(* IEC 61131-3 sources: scada_scout/plc_programs (part 2) *)

(* ---- PRG_GPS01GPC02UPM01FCB02.st ---- *)
(* ========================================================================
   PLC PROGRAM: PRG_GPS01GPC02UPM01FCB02
   IED: GPS01GPC02UPM01FCB02
   Device: GPS01GPC02UPM01FCB02
   Generated: 2026-02-05 10:47:33

   This program runs cyclically (default 100ms) and has access to all
   data points of the associated IEC 61850 device. Users can add custom
   logic in the designated sections below.
   ======================================================================== *)

PROGRAM PRG_GPS01GPC02UPM01FCB02
VAR
    (* ====== System Variables ====== *)
    cycle_count: UDINT := 0;           (* Increments each scan cycle *)
    first_scan: BOOL := TRUE;          (* TRUE only on first execution *)
    scan_time_ms: REAL := 0.0;         (* Last scan time in milliseconds *)

    (* ====== IED Connection Status ====== *)
    ied_connected: BOOL := FALSE;      (* TRUE when IED server is running *)
    ied_name: STRING := 'GPS01GPC02UPM01FCB02';
    device_name: STRING := 'GPS01GPC02UPM01FCB02';

    (* ====== Logical Devices ====== *)
    (* Available LDs: AnUn_ArcProtInput1, Application, BinIO, BinIO_BinaryInputs, BinIO_BinaryOutputs, CB1, CB1_Fundamental, Ds1, Ds2, Mod1, Mod1_Channel1, Mod2, Mod2_Channel1, Mod3, Mod3_Channel1, PowS, PowS_MeasPointI3ph1, PowS_MeasPointV3ph1, Rec, Rec_FaultRecorder, VI3p1, VI3p1_5051NOCgndB1, VI3p1_5051OC3phase1, VI3p1_ArcProtection1, VI3p1_Energy, VI3p1_FundSymComp, VI3p1_OperationalValues, VI3p1_ProcessMonitor, VI3p1_ExternalTrip1, VI3p1_67DirOC3phB1, VI3p1_67NDirOCgndB1, ComSupervision, ComSupervision_GOOSE *)

    (* ====== User Variables ====== *)
    (* Add your custom variables here *)
    (* Example:
    timer1: TON;
    counter: INT := 0;
    status_word: WORD;
    *)

END_VAR

(* ======================================================================
   INITIALIZATION SECTION
   Runs once on first scan. Use for setup and initialization.
   ====================================================================== *)
IF first_scan THEN
    (* Initialize user variables here *)
    cycle_count := 0;

    (* Log program start *)
    (* SCADA_LOG('INFO', CONCAT('PLC Program started: ', device_name)); *)

    first_scan := FALSE;
END_IF;

(* ======================================================================
   MAIN CYCLIC EXECUTION
   This section runs continuously every scan cycle (default 100ms).
   ====================================================================== *)

(* Increment cycle counter *)
cycle_count := cycle_count + 1;

(* ====== USER LOGIC SECTION 1: Pre-Processing ====== *)
(* Add logic that should run before main processing *)
(* Example:
IF ied_connected THEN
    (* Read IED data points *)
    (* status_word := READ_IED_DATA(device_name, 'LD0/MMXU1$MX$TotW$mag'); *)
END_IF;
*)

(* ====== USER LOGIC SECTION 2: Main Processing ====== *)
(* Add your main control logic here *)
(* Example:
IF counter > 100 THEN
    counter := 0;
    (* Perform periodic action *)
END_IF;
counter := counter + 1;
*)

(* ====== USER LOGIC SECTION 3: Post-Processing ====== *)
(* Add logic for outputs, writes, and cleanup *)
(* Example:
IF ied_connected THEN
    (* Write control commands to IED *)
    (* WRITE_IED_CONTROL(device_name, 'LD0/CSWI1$CO$Pos', TRUE); *)
END_IF;
*)

(* ====== Built-in Functions Available ====== *)
(*
   READ_IED_DATA(device: STRING, ref: STRING): ANY
       - Read data from IED object reference
       - Example: READ_IED_DATA('MyIED', 'LD0/MMXU1$MX$TotW$mag')

   WRITE_IED_DATA(device: STRING, ref: STRING, value: ANY): BOOL
       - Write data to IED object reference
       - Returns TRUE on success

   WRITE_IED_CONTROL(device: STRING, ref: STRING, value: ANY): BOOL
       - Send control command to IED
       - Returns TRUE on success

   SCADA_LOG(level: STRING, message: STRING)
       - Log message to event log
       - Levels: 'INFO', 'WARNING', 'ERROR'

   GET_DEVICE_STATUS(device: STRING): BOOL
       - Check if device is connected
*)

END_PROGRAM

(* ---- PRG_GPS01GPC02UPM01MCB01.st ---- *)
(* ========================================================================
   PLC PROGRAM: PRG_GPS01GPC02UPM01MCB01
   IED: GPS01GPC02UPM01MCB01
   Device: GPS01GPC02UPM01MCB01
   Generated: 2026-02-05 10:47:34

   This program runs cyclically (default 100ms) and has access to all
   data points of the associated IEC 61850 device. Users can add custom
   logic in the designated sections below.
   ======================================================================== *)

PROGRAM PRG_GPS01GPC02UPM01MCB01
VAR
    (* ====== System Variables ====== *)
    cycle_count: UDINT := 0;           (* Increments each scan cycle *)
    first_scan: BOOL := TRUE;          (* TRUE only on first execution *)
    scan_time_ms: REAL := 0.0;         (* Last scan time in milliseconds *)

    (* ====== IED Connection Status ====== *)
    ied_connected: BOOL := FALSE;      (* TRUE when IED server is running *)
    ied_name: STRING := 'GPS01GPC02UPM01MCB01';
    device_name: STRING := 'GPS01GPC02UPM01MCB01';

    (* ====== Logical Devices ====== *)
    (* Available LDs: AnUn_ArcProtInput1, Application, BinIO, BinIO_BinaryInputs, BinIO_BinaryOutputs, CB1, CB1_Fundamental, Ds1, Ds2, Mod1, Mod1_Channel1, Mod2, Mod2_Channel1, Mod3, Mod3_Channel1, PowS, PowS_MeasPointI3ph1, PowS_MeasPointV3ph1, Rec, Rec_FaultRecorder, VI3p1, VI3p1_5051NOCgndB1, VI3p1_5051OC3phase1, VI3p1_ArcProtection1, VI3p1_Energy, VI3p1_FundSymComp, VI3p1_OperationalValues, VI3p1_ProcessMonitor, VI3p1_ExternalTrip1, VI3p1_67DirOC3phB1, VI3p1_67NDirOCgndB1, VI3p1_ExternalTrip2, ComSupervision, ComSupervision_GOOSE *)

    (* ====== User Variables ====== *)
    (* Add your custom variables here *)
    (* Example:
    timer1: TON;
    counter: INT := 0;
    status_word: WORD;
    *)

END_VAR

(* ======================================================================
   INITIALIZATION SECTION
   Runs once on first scan. Use for setup and initialization.
   ====================================================================== *)
IF first_scan THEN
    (* Initialize user variables here *)
    cycle_count := 0;

    (* Log program start *)
    (* SCADA_LOG('INFO', CONCAT('PLC Program started: ', device_name)); *)

    first_scan := FALSE;
END_IF;

(* ======================================================================
   MAIN CYCLIC EXECUTION
   This section runs continuously every scan cycle (default 100ms).
   ====================================================================== *)

(* Increment cycle counter *)
cycle_count := cycle_count + 1;

(* ====== USER LOGIC SECTION 1: Pre-Processing ====== *)
(* Add logic that should run before main processing *)
(* Example:
IF ied_connected THEN
    (* Read IED data points *)
    (* status_word := READ_IED_DATA(device_name, 'LD0/MMXU1$MX$TotW$mag'); *)
END_IF;
*)

(* ====== USER LOGIC SECTION 2: Main Processing ====== *)
(* Add your main control logic here *)
(* Example:
IF counter > 100 THEN
    counter := 0;
    (* Perform periodic action *)
END_IF;
counter := counter + 1;
*)

(* ====== USER LOGIC SECTION 3: Post-Processing ====== *)
(* Add logic for outputs, writes, and cleanup *)
(* Example:
IF ied_connected THEN
    (* Write control commands to IED *)
    (* WRITE_IED_CONTROL(device_name, 'LD0/CSWI1$CO$Pos', TRUE); *)
END_IF;
*)

(* ====== Built-in Functions Available ====== *)
(*
   READ_IED_DATA(device: STRING, ref: STRING): ANY
       - Read data from IED object reference
       - Example: READ_IED_DATA('MyIED', 'LD0/MMXU1$MX$TotW$mag')

   WRITE_IED_DATA(device: STRING, ref: STRING, value: ANY): BOOL
       - Write data to IED object reference
       - Returns TRUE on success

   WRITE_IED_CONTROL(device: STRING, ref: STRING, value: ANY): BOOL
       - Send control command to IED
       - Returns TRUE on success

   SCADA_LOG(level: STRING, message: STRING)
       - Log message to event log
       - Levels: 'INFO', 'WARNING', 'ERROR'

   GET_DEVICE_STATUS(device: STRING): BOOL
       - Check if device is connected
*)

END_PROGRAM

(* ---- PRG_GPS01GPC03UPM01FCB01.st ---- *)
(* ========================================================================
   PLC PROGRAM: PRG_GPS01GPC03UPM01FCB01
   IED: GPS01GPC03UPM01FCB01
   Device: GPS01GPC03UPM01FCB01
   Generated: 2026-02-05 10:47:34

   This program runs cyclically (default 100ms) and has access to all
   data points of the associated IEC 61850 device. Users can add custom
   logic in the designated sections below.
   ======================================================================== *)

PROGRAM PRG_GPS01GPC03UPM01FCB01
VAR
    (* ====== System Variables ====== *)
    cycle_count: UDINT := 0;           (* Increments each scan cycle *)
    first_scan: BOOL := TRUE;          (* TRUE only on first execution *)
    scan_time_ms: REAL := 0.0;         (* Last scan time in milliseconds *)

    (* ====== IED Connection Status ====== *)
    ied_connected: BOOL := FALSE;      (* TRUE when IED server is running *)
    ied_name: STRING := 'GPS01GPC03UPM01FCB01';
    device_name: STRING := 'GPS01GPC03UPM01FCB01';

    (* ====== Logical Devices ====== *)
    (* Available LDs: AnUn_ArcProtInput1, Application, BinIO, BinIO_BinaryInputs, BinIO_BinaryOutputs, CB1, CB1_Fundamental, Ds1, Ds2, Mod1, Mod1_Channel1, Mod2, Mod2_Channel1, Mod3, Mod3_Channel1, PowS, PowS_MeasPointI3ph1, PowS_MeasPointV3ph1, Rec, Rec_FaultRecorder, VI3p1, VI3p1_5051NOCgndB1, VI3p1_5051OC3phase1, VI3p1_ArcProtection1, VI3p1_Energy, VI3p1_FundSymComp, VI3p1_OperationalValues, VI3p1_ProcessMonitor, VI3p1_ExternalTrip1, VI3p1_67DirOC3phB1, VI3p1_67NDirOCgndB1, ComSupervision, ComSupervision_GOOSE *)

    (* ====== User Variables ====== *)
    (* Add your custom variables here *)
    (* Example:
    timer1: TON;
    counter: INT := 0;
    status_word: WORD;
    *)

END_VAR

(* ======================================================================
   INITIALIZATION SECTION
   Runs once on first scan. Use for setup and initialization.
   ====================================================================== *)
IF first_scan THEN
    (* Initialize user variables here *)
    cycle_count := 0;

    (* Log program start *)
    (* SCADA_LOG('INFO', CONCAT('PLC Program started: ', device_name)); *)

    first_scan := FALSE;
END_IF;

(* ======================================================================
   MAIN CYCLIC EXECUTION
   This section runs continuously every scan cycle (default 100ms).
   ====================================================================== *)

(* Increment cycle counter *)
cycle_count := cycle_count + 1;

(* ====== USER LOGIC SECTION 1: Pre-Processing ====== *)
(* Add logic that should run before main processing *)
(* Example:
IF ied_connected THEN
    (* Read IED data points *)
    (* status_word := READ_IED_DATA(device_name, 'LD0/MMXU1$MX$TotW$mag'); *)
END_IF;
*)

(* ====== USER LOGIC SECTION 2: Main Processing ====== *)
(* Add your main control logic here *)
(* Example:
IF counter > 100 THEN
    counter := 0;
    (* Perform periodic action *)
END_IF;
counter := counter + 1;
*)

(* ====== USER LOGIC SECTION 3: Post-Processing ====== *)
(* Add logic for outputs, writes, and cleanup *)
(* Example:
IF ied_connected THEN
    (* Write control commands to IED *)
    (* WRITE_IED_CONTROL(device_name, 'LD0/CSWI1$CO$Pos', TRUE); *)
END_IF;
*)

(* ====== Built-in Functions Available ====== *)
(*
   READ_IED_DATA(device: STRING, ref: STRING): ANY
       - Read data from IED object reference
       - Example: READ_IED_DATA('MyIED', 'LD0/MMXU1$MX$TotW$mag')

   WRITE_IED_DATA(device: STRING, ref: STRING, value: ANY): BOOL
       - Write data to IED object reference
       - Returns TRUE on success

   WRITE_IED_CONTROL(device: STRING, ref: STRING, value: ANY): BOOL
       - Send control command to IED
       - Returns TRUE on success

   SCADA_LOG(level: STRING, message: STRING)
       - Log message to event log
       - Levels: 'INFO', 'WARNING', 'ERROR'

   GET_DEVICE_STATUS(device: STRING): BOOL
       - Check if device is connected
*)

END_PROGRAM

(* ---- PRG_GPS01GPC03UPM01FCB02.st ---- *)
(* ========================================================================
   PLC PROGRAM: PRG_GPS01GPC03UPM01FCB02
   IED: GPS01GPC03UPM01FCB02
   Device: GPS01GPC03UPM01FCB02
   Generated: 2026-02-05 10:47:35

   This program runs cyclically (default 100ms) and has access to all
   data points of the associated IEC 61850 device. Users can add custom
   logic in the designated sections below.
   ======================================================================== *)

PROGRAM PRG_GPS01GPC03UPM01FCB02
VAR
    (* ====== System Variables ====== *)
    cycle_count: UDINT := 0;           (* Increments each scan cycle *)
    first_scan: BOOL := TRUE;          (* TRUE only on first execution *)
    scan_time_ms: REAL := 0.0;         (* Last scan time in milliseconds *)

    (* ====== IED Connection Status ====== *)
    ied_connected: BOOL := FALSE;      (* TRUE when IED server is running *)
    ied_name: STRING := 'GPS01GPC03UPM01FCB02';
    device_name: STRING := 'GPS01GPC03UPM01FCB02';

    (* ====== Logical Devices ====== *)
    (* Available LDs: AnUn_ArcProtInput1, Application, BinIO, BinIO_BinaryInputs, BinIO_BinaryOutputs, CB1, CB1_Fundamental, Ds1, Ds2, Mod1, Mod1_Channel1, Mod2, Mod2_Channel1, Mod3, Mod3_Channel1, PowS, PowS_MeasPointI3ph1, PowS_MeasPointV3ph1, Rec, Rec_FaultRecorder, VI3p1, VI3p1_5051NOCgndB1, VI3p1_5051OC3phase1, VI3p1_ArcProtection1, VI3p1_Energy, VI3p1_FundSymComp, VI3p1_OperationalValues, VI3p1_ProcessMonitor, VI3p1_ExternalTrip1, VI3p1_67DirOC3phB1, VI3p1_67NDirOCgndB1, ComSupervision, ComSupervision_GOOSE *)

    (* ====== User Variables ====== *)
    (* Add your custom variables here *)
    (* Example:
    timer1: TON;
    counter: INT := 0;
    status_word: WORD;
    *)

END_VAR

(* ======================================================================
   INITIALIZATION SECTION
   Runs once on first scan. Use for setup and initialization.
   ====================================================================== *)
IF first_scan THEN
    (* Initialize user variables here *)
    cycle_count := 0;

    (* Log program start *)
    (* SCADA_LOG('INFO', CONCAT('PLC Program started: ', device_name)); *)

    first_scan := FALSE;
END_IF;

(* ======================================================================
   MAIN CYCLIC EXECUTION
   This section runs continuously every scan cycle (default 100ms).
   ====================================================================== *)

(* Increment cycle counter *)
cycle_count := cycle_count + 1;

(* ====== USER LOGIC SECTION 1: Pre-Processing ====== *)
(* Add logic that should run before main processing *)
(* Example:
IF ied_connected THEN
    (* Read IED data points *)
    (* status_word := READ_IED_DATA(device_name, 'LD0/MMXU1$MX$TotW$mag'); *)
END_IF;
*)

(* ====== USER LOGIC SECTION 2: Main Processing ====== *)
(* Add your main control logic here *)
(* Example:
IF counter > 100 THEN
    counter := 0;
    (* Perform periodic action *)
END_IF;
counter := counter + 1;
*)

(* ====== USER LOGIC SECTION 3: Post-Processing ====== *)
(* Add logic for outputs, writes, and cleanup *)
(* Example:
IF ied_connected THEN
    (* Write control commands to IED *)
    (* WRITE_IED_CONTROL(device_name, 'LD0/CSWI1$CO$Pos', TRUE); *)
END_IF;
*)

(* ====== Built-in Functions Available ====== *)
(*
   READ_IED_DATA(device: STRING, ref: STRING): ANY
       - Read data from IED object reference
       - Example: READ_IED_DATA('MyIED', 'LD0/MMXU1$MX$TotW$mag')

   WRITE_IED_DATA(device: STRING, ref: STRING, value: ANY): BOOL
       - Write data to IED object reference
       - Returns TRUE on success

   WRITE_IED_CONTROL(device: STRING, ref: STRING, value: ANY): BOOL
       - Send control command to IED
       - Returns TRUE on success

   SCADA_LOG(level: STRING, message: STRING)
       - Log message to event log
       - Levels: 'INFO', 'WARNING', 'ERROR'

   GET_DEVICE_STATUS(device: STRING): BOOL
       - Check if device is connected
*)

END_PROGRAM

(* ---- PRG_GPS01GPC03UPM01MCB01.st ---- *)
(* ========================================================================
   PLC PROGRAM: PRG_GPS01GPC03UPM01MCB01
   IED: GPS01GPC03UPM01MCB01
   Device: GPS01GPC03UPM01MCB01
   Generated: 2026-02-05 10:47:36

   This program runs cyclically (default 100ms) and has access to all
   data points of the associated IEC 61850 device. Users can add custom
   logic in the designated sections below.
   ======================================================================== *)

PROGRAM PRG_GPS01GPC03UPM01MCB01
VAR
    (* ====== System Variables ====== *)
    cycle_count: UDINT := 0;           (* Increments each scan cycle *)
    first_scan: BOOL := TRUE;          (* TRUE only on first execution *)
    scan_time_ms: REAL := 0.0;         (* Last scan time in milliseconds *)

    (* ====== IED Connection Status ====== *)
    ied_connected: BOOL := FALSE;      (* TRUE when IED server is running *)
    ied_name: STRING := 'GPS01GPC03UPM01MCB01';
    device_name: STRING := 'GPS01GPC03UPM01MCB01';

    (* ====== Logical Devices ====== *)
    (* Available LDs: AnUn_ArcProtInput1, Application, BinIO, BinIO_BinaryInputs, BinIO_BinaryOutputs, CB1, CB1_Fundamental, Ds1, Ds2, Mod1, Mod1_Channel1, Mod2, Mod2_Channel1, Mod3, Mod3_Channel1, PowS, PowS_MeasPointI3ph1, PowS_MeasPointV3ph1, Rec, Rec_FaultRecorder, VI3p1, VI3p1_5051NOCgndB1, VI3p1_5051OC3phase1, VI3p1_ArcProtection1, VI3p1_Energy, VI3p1_FundSymComp, VI3p1_OperationalValues, VI3p1_ProcessMonitor, VI3p1_67DirOC3phB1, VI3p1_ExternalTrip1, VI3p1_67NDirOCgndB1, VI3p1_ExternalTrip2, ComSupervision, ComSupervision_GOOSE *)

    (* ====== User Variables ====== *)
    (* Add your custom variables here *)
    (* Example:
    timer1: TON;
    counter: INT := 0;
    status_word: WORD;
    *)

END_VAR

(* ======================================================================
   INITIALIZATION SECTION
   Runs once on first scan. Use for setup and initialization.
   ====================================================================== *)
IF first_scan THEN
    (* Initialize user variables here *)
    cycle_count := 0;

    (* Log program start *)
    (* SCADA_LOG('INFO', CONCAT('PLC Program started: ', device_name)); *)

    first_scan := FALSE;
END_IF;

(* ======================================================================
   MAIN CYCLIC EXECUTION
   This section runs continuously every scan cycle (default 100ms).
   ====================================================================== *)

(* Increment cycle counter *)
cycle_count := cycle_count + 1;

(* ====== USER LOGIC SECTION 1: Pre-Processing ====== *)
(* Add logic that should run before main processing *)
(* Example:
IF ied_connected THEN
    (* Read IED data points *)
    (* status_word := READ_IED_DATA(device_name, 'LD0/MMXU1$MX$TotW$mag'); *)
END_IF;
*)

(* ====== USER LOGIC SECTION 2: Main Processing ====== *)
(* Add your main control logic here *)
(* Example:
IF counter > 100 THEN
    counter := 0;
    (* Perform periodic action *)
END_IF;
counter := counter + 1;
*)

(* ====== USER LOGIC SECTION 3: Post-Processing ====== *)
(* Add logic for outputs, writes, and cleanup *)
(* Example:
IF ied_connected THEN
    (* Write control commands to IED *)
    (* WRITE_IED_CONTROL(device_name, 'LD0/CSWI1$CO$Pos', TRUE); *)
END_IF;
*)

(* ====== Built-in Functions Available ====== *)
(*
   READ_IED_DATA(device: STRING, ref: STRING): ANY
       - Read data from IED object reference
       - Example: READ_IED_DATA('MyIED', 'LD0/MMXU1$MX$TotW$mag')

   WRITE_IED_DATA(device: STRING, ref: STRING, value: ANY): BOOL
       - Write data to IED object reference
       - Returns TRUE on success

   WRITE_IED_CONTROL(device: STRING, ref: STRING, value: ANY): BOOL
       - Send control command to IED
       - Returns TRUE on success

   SCADA_LOG(level: STRING, message: STRING)
       - Log message to event log
       - Levels: 'INFO', 'WARNING', 'ERROR'

   GET_DEVICE_STATUS(device: STRING): BOOL
       - Check if device is connected
*)

END_PROGRAM

(* ---- PRG_GPS01GPC04UPM01FCB01.st ---- *)
(* ========================================================================
   PLC PROGRAM: PRG_GPS01GPC04UPM01FCB01
   IED: GPS01GPC04UPM01FCB01
   Device: GPS01GPC04UPM01FCB01
   Generated: 2026-02-05 10:47:36

   This program runs cyclically (default 100ms) and has access to all
   data points of the associated IEC 61850 device. Users can add custom
   logic in the designated sections below.
   ======================================================================== *)

PROGRAM PRG_GPS01GPC04UPM01FCB01
VAR
    (* ====== System Variables ====== *)
    cycle_count: UDINT := 0;           (* Increments each scan cycle *)
    first_scan: BOOL := TRUE;          (* TRUE only on first execution *)
    scan_time_ms: REAL := 0.0;         (* Last scan time in milliseconds *)

    (* ====== IED Connection Status ====== *)
    ied_connected: BOOL := FALSE;      (* TRUE when IED server is running *)
    ied_name: STRING := 'GPS01GPC04UPM01FCB01';
    device_name: STRING := 'GPS01GPC04UPM01FCB01';

    (* ====== Logical Devices ====== *)
    (* Available LDs: AnUn_ArcProtInput1, Application, BinIO, BinIO_BinaryInputs, BinIO_BinaryOutputs, CB1, CB1_Fundamental, Ds1, Ds2, Mod1, Mod1_Channel1, Mod2, Mod2_Channel1, Mod3, Mod3_Channel1, PowS, PowS_MeasPointI3ph1, PowS_MeasPointV3ph1, Rec, Rec_FaultRecorder, VI3p1, VI3p1_5051NOCgndB1, VI3p1_5051OC3phase1, VI3p1_ArcProtection1, VI3p1_Energy, VI3p1_FundSymComp, VI3p1_OperationalValues, VI3p1_ProcessMonitor, VI3p1_ExternalTrip1, VI3p1_67DirOC3phB1, VI3p1_67NDirOCgndB1, ComSupervision, ComSupervision_GOOSE *)

    (* ====== User Variables ====== *)
    (* Add your custom variables here *)
    (* Example:
    timer1: TON;
    counter: INT := 0;
    status_word: WORD;
    *)

END_VAR

(* ======================================================================
   INITIALIZATION SECTION
   Runs once on first scan. Use for setup and initialization.
   ====================================================================== *)
IF first_scan THEN
    (* Initialize user variables here *)
    cycle_count := 0;

    (* Log program start *)
    (* SCADA_LOG('INFO', CONCAT('PLC Program started: ', device_name)); *)

    first_scan := FALSE;
END_IF;

(* ======================================================================
   MAIN CYCLIC EXECUTION
   This section runs continuously every scan cycle (default 100ms).
   ====================================================================== *)

(* Increment cycle counter *)
cycle_count := cycle_count + 1;

(* ====== USER LOGIC SECTION 1: Pre-Processing ====== *)
(* Add logic that should run before main processing *)
(* Example:
IF ied_connected THEN
    (* Read IED data points *)
    (* status_word := READ_IED_DATA(device_name, 'LD0/MMXU1$MX$TotW$mag'); *)
END_IF;
*)

(* ====== USER LOGIC SECTION 2: Main Processing ====== *)
(* Add your main control logic here *)
(* Example:
IF counter > 100 THEN
    counter := 0;
    (* Perform periodic action *)
END_IF;
counter := counter + 1;
*)

(* ====== USER LOGIC SECTION 3: Post-Processing ====== *)
(* Add logic for outputs, writes, and cleanup *)
(* Example:
IF ied_connected THEN
    (* Write control commands to IED *)
    (* WRITE_IED_CONTROL(device_name, 'LD0/CSWI1$CO$Pos', TRUE); *)
END_IF;
*)

(* ====== Built-in Functions Available ====== *)
(*
   READ_IED_DATA(device: STRING, ref: STRING): ANY
       - Read data from IED object reference
       - Example: READ_IED_DATA('MyIED', 'LD0/MMXU1$MX$TotW$mag')

   WRITE_IED_DATA(device: STRING, ref: STRING, value: ANY): BOOL
       - Write data to IED object reference
       - Returns TRUE on success

   WRITE_IED_CONTROL(device: STRING, ref: STRING, value: ANY): BOOL
       - Send control command to IED
       - Returns TRUE on success

   SCADA_LOG(level: STRING, message: STRING)
       - Log message to event log
       - Levels: 'INFO', 'WARNING', 'ERROR'

   GET_DEVICE_STATUS(device: STRING): BOOL
       - Check if device is connected
*)

END_PROGRAM

(* ---- PRG_GPS01GPC04UPM01FCB02.st ---- *)
(* ========================================================================
   PLC PROGRAM: PRG_GPS01GPC04UPM01FCB02
   IED: GPS01GPC04UPM01FCB02
   Device: GPS01GPC04UPM01FCB02
   Generated: 2026-02-05 10:47:38

   This program runs cyclically (default 100ms) and has access to all
   data points of the associated IEC 61850 device. Users can add custom
   logic in the designated sections below.
   ======================================================================== *)

PROGRAM PRG_GPS01GPC04UPM01FCB02
VAR
    (* ====== System Variables ====== *)
    cycle_count: UDINT := 0;           (* Increments each scan cycle *)
    first_scan: BOOL := TRUE;          (* TRUE only on first execution *)
    scan_time_ms: REAL := 0.0;         (* Last scan time in milliseconds *)

    (* ====== IED Connection Status ====== *)
    ied_connected: BOOL := FALSE;      (* TRUE when IED server is running *)
    ied_name: STRING := 'GPS01GPC04UPM01FCB02';
    device_name: STRING := 'GPS01GPC04UPM01FCB02';

    (* ====== Logical Devices ====== *)
    (* Available LDs: AnUn_ArcProtInput1, Application, BinIO, BinIO_BinaryInputs, BinIO_BinaryOutputs, CB1, CB1_Fundamental, Ds1, Ds2, Mod1, Mod1_Channel1, Mod2, Mod2_Channel1, Mod3, Mod3_Channel1, PowS, PowS_MeasPointI3ph1, PowS_MeasPointV3ph1, Rec, Rec_FaultRecorder, VI3p1, VI3p1_5051NOCgndB1, VI3p1_5051OC3phase1, VI3p1_ArcProtection1, VI3p1_Energy, VI3p1_FundSymComp, VI3p1_OperationalValues, VI3p1_ProcessMonitor, VI3p1_ExternalTrip1, VI3p1_67DirOC3phB1, VI3p1_67NDirOCgndB1, ComSupervision, ComSupervision_GOOSE *)

    (* ====== User Variables ====== *)
    (* Add your custom variables here *)
    (* Example:
    timer1: TON;
    counter: INT := 0;
    status_word: WORD;
    *)

END_VAR

(* ======================================================================
   INITIALIZATION SECTION
   Runs once on first scan. Use for setup and initialization.
   ====================================================================== *)
IF first_scan THEN
    (* Initialize user variables here *)
    cycle_count := 0;

    (* Log program start *)
    (* SCADA_LOG('INFO', CONCAT('PLC Program started: ', device_name)); *)

    first_scan := FALSE;
END_IF;

(* ======================================================================
   MAIN CYCLIC EXECUTION
   This section runs continuously every scan cycle (default 100ms).
   ====================================================================== *)

(* Increment cycle counter *)
cycle_count := cycle_count + 1;

(* ====== USER LOGIC SECTION 1: Pre-Processing ====== *)
(* Add logic that should run before main processing *)
(* Example:
IF ied_connected THEN
    (* Read IED data points *)
    (* status_word := READ_IED_DATA(device_name, 'LD0/MMXU1$MX$TotW$mag'); *)
END_IF;
*)

(* ====== USER LOGIC SECTION 2: Main Processing ====== *)
(* Add your main control logic here *)
(* Example:
IF counter > 100 THEN
    counter := 0;
    (* Perform periodic action *)
END_IF;
counter := counter + 1;
*)

(* ====== USER LOGIC SECTION 3: Post-Processing ====== *)
(* Add logic for outputs, writes, and cleanup *)
(* Example:
IF ied_connected THEN
    (* Write control commands to IED *)
    (* WRITE_IED_CONTROL(device_name, 'LD0/CSWI1$CO$Pos', TRUE); *)
END_IF;
*)

(* ====== Built-in Functions Available ====== *)
(*
   READ_IED_DATA(device: STRING, ref: STRING): ANY
       - Read data from IED object reference
       - Example: READ_IED_DATA('MyIED', 'LD0/MMXU1$MX$TotW$mag')

   WRITE_IED_DATA(device: STRING, ref: STRING, value: ANY): BOOL
       - Write data to IED object reference
       - Returns TRUE on success

   WRITE_IED_CONTROL(device: STRING, ref: STRING, value: ANY): BOOL
       - Send control command to IED
       - Returns TRUE on success

   SCADA_LOG(level: STRING, message: STRING)
       - Log message to event log
       - Levels: 'INFO', 'WARNING', 'ERROR'

   GET_DEVICE_STATUS(device: STRING): BOOL
       - Check if device is connected
*)

END_PROGRAM

(* ---- PRG_GPS01GPC04UPM01MCB01.st ---- *)
(* ========================================================================
   PLC PROGRAM: PRG_GPS01GPC04UPM01MCB01
   IED: GPS01GPC04UPM01MCB01
   Device: GPS01GPC04UPM01MCB01
   Generated: 2026-02-05 10:47:39

   This program runs cyclically (default 100ms) and has access to all
   data points of the associated IEC 61850 device. Users can add custom
   logic in the designated sections below.
   ======================================================================== *)

PROGRAM PRG_GPS01GPC04UPM01MCB01
VAR
    (* ====== System Variables ====== *)
    cycle_count: UDINT := 0;           (* Increments each scan cycle *)
    first_scan: BOOL := TRUE;          (* TRUE only on first execution *)
    scan_time_ms: REAL := 0.0;         (* Last scan time in milliseconds *)

    (* ====== IED Connection Status ====== *)
    ied_connected: BOOL := FALSE;      (* TRUE when IED server is running *)
    ied_name: STRING := 'GPS01GPC04UPM01MCB01';
    device_name: STRING := 'GPS01GPC04UPM01MCB01';

    (* ====== Logical Devices ====== *)
    (* Available LDs: AnUn_ArcProtInput1, Application, BinIO, BinIO_BinaryInputs, BinIO_BinaryOutputs, CB1, CB1_Fundamental, Ds1, Ds2, Mod1, Mod1_Channel1, Mod2, Mod2_Channel1, Mod3, Mod3_Channel1, PowS, PowS_MeasPointI3ph1, PowS_MeasPointV3ph1, Rec, Rec_FaultRecorder, VI3p1, VI3p1_5051NOCgndB1, VI3p1_5051OC3phase1, VI3p1_ArcProtection1, VI3p1_Energy, VI3p1_FundSymComp, VI3p1_OperationalValues, VI3p1_ProcessMonitor, VI3p1_ExternalTrip1, VI3p1_67DirOC3phB1, VI3p1_67NDirOCgndB1, VI3p1_ExternalTrip2, ComSupervision, ComSupervision_GOOSE *)

    (* ====== User Variables ====== *)
    (* Add your custom variables here *)
    (* Example:
    timer1: TON;
    counter: INT := 0;
    status_word: WORD;
    *)

END_VAR

(* ======================================================================
   INITIALIZATION SECTION
   Runs once on first scan. Use for setup and initialization.
   ====================================================================== *)
IF first_scan THEN
    (* Initialize user variables here *)
    cycle_count := 0;

    (* Log program start *)
    (* SCADA_LOG('INFO', CONCAT('PLC Program started: ', device_name)); *)

    first_scan := FALSE;
END_IF;

(* ======================================================================
   MAIN CYCLIC EXECUTION
   This section runs continuously every scan cycle (default 100ms).
   ====================================================================== *)

(* Increment cycle counter *)
cycle_count := cycle_count + 1;

(* ====== USER LOGIC SECTION 1: Pre-Processing ====== *)
(* Add logic that should run before main processing *)
(* Example:
IF ied_connected THEN
    (* Read IED data points *)
    (* status_word := READ_IED_DATA(device_name, 'LD0/MMXU1$MX$TotW$mag'); *)
END_IF;
*)

(* ====== USER LOGIC SECTION 2: Main Processing ====== *)
(* Add your main control logic here *)
(* Example:
IF counter > 100 THEN
    counter := 0;
    (* Perform periodic action *)
END_IF;
counter := counter + 1;
*)

(* ====== USER LOGIC SECTION 3: Post-Processing ====== *)
(* Add logic for outputs, writes, and cleanup *)
(* Example:
IF ied_connected THEN
    (* Write control commands to IED *)
    (* WRITE_IED_CONTROL(device_name, 'LD0/CSWI1$CO$Pos', TRUE); *)
END_IF;
*)

(* ====== Built-in Functions Available ====== *)
(*
   READ_IED_DATA(device: STRING, ref: STRING): ANY
       - Read data from IED object reference
       - Example: READ_IED_DATA('MyIED', 'LD0/MMXU1$MX$TotW$mag')

   WRITE_IED_DATA(device: STRING, ref: STRING, value: ANY): BOOL
       - Write data to IED object reference
       - Returns TRUE on success

   WRITE_IED_CONTROL(device: STRING, ref: STRING, value: ANY): BOOL
       - Send control command to IED
       - Returns TRUE on success

   SCADA_LOG(level: STRING, message: STRING)
       - Log message to event log
       - Levels: 'INFO', 'WARNING', 'ERROR'

   GET_DEVICE_STATUS(device: STRING): BOOL
       - Check if device is connected
*)

END_PROGRAM

(* ---- PRG_GPS01GPC05UPM01FCB01.st ---- *)
(* ========================================================================
   PLC PROGRAM: PRG_GPS01GPC05UPM01FCB01
   IED: GPS01GPC05UPM01FCB01
   Device: GPS01GPC05UPM01FCB01
   Generated: 2026-02-05 10:47:39

   This program runs cyclically (default 100ms) and has access to all
   data points of the associated IEC 61850 device. Users can add custom
   logic in the designated sections below.
   ======================================================================== *)

PROGRAM PRG_GPS01GPC05UPM01FCB01
VAR
    (* ====== System Variables ====== *)
    cycle_count: UDINT := 0;           (* Increments each scan cycle *)
    first_scan: BOOL := TRUE;          (* TRUE only on first execution *)
    scan_time_ms: REAL := 0.0;         (* Last scan time in milliseconds *)

    (* ====== IED Connection Status ====== *)
    ied_connected: BOOL := FALSE;      (* TRUE when IED server is running *)
    ied_name: STRING := 'GPS01GPC05UPM01FCB01';
    device_name: STRING := 'GPS01GPC05UPM01FCB01';

    (* ====== Logical Devices ====== *)
    (* Available LDs: AnUn_ArcProtInput1, Application, BinIO, BinIO_BinaryInputs, BinIO_BinaryOutputs, CB1, CB1_Fundamental, Ds1, Ds2, Mod1, Mod1_Channel1, Mod2, Mod2_Channel1, Mod3, Mod3_Channel1, PowS, PowS_MeasPointI3ph1, PowS_MeasPointV3ph1, Rec, Rec_FaultRecorder, VI3p1, VI3p1_5051NOCgndB1, VI3p1_5051OC3phase1, VI3p1_ArcProtection1, VI3p1_Energy, VI3p1_FundSymComp, VI3p1_OperationalValues, VI3p1_ProcessMonitor, VI3p1_ExternalTrip1, VI3p1_67DirOC3phB1, VI3p1_67NDirOCgndB1, ComSupervision, ComSupervision_GOOSE *)

    (* ====== User Variables ====== *)
    (* Add your custom variables here *)
    (* Example:
    timer1: TON;
    counter: INT := 0;
    status_word: WORD;
    *)

END_VAR

(* ======================================================================
   INITIALIZATION SECTION
   Runs once on first scan. Use for setup and initialization.
   ====================================================================== *)
IF first_scan THEN
    (* Initialize user variables here *)
    cycle_count := 0;

    (* Log program start *)
    (* SCADA_LOG('INFO', CONCAT('PLC Program started: ', device_name)); *)

    first_scan := FALSE;
END_IF;

(* ======================================================================
   MAIN CYCLIC EXECUTION
   This section runs continuously every scan cycle (default 100ms).
   ====================================================================== *)

(* Increment cycle counter *)
cycle_count := cycle_count + 1;

(* ====== USER LOGIC SECTION 1: Pre-Processing ====== *)
(* Add logic that should run before main processing *)
(* Example:
IF ied_connected THEN
    (* Read IED data points *)
    (* status_word := READ_IED_DATA(device_name, 'LD0/MMXU1$MX$TotW$mag'); *)
END_IF;
*)

(* ====== USER LOGIC SECTION 2: Main Processing ====== *)
(* Add your main control logic here *)
(* Example:
IF counter > 100 THEN
    counter := 0;
    (* Perform periodic action *)
END_IF;
counter := counter + 1;
*)

(* ====== USER LOGIC SECTION 3: Post-Processing ====== *)
(* Add logic for outputs, writes, and cleanup *)
(* Example:
IF ied_connected THEN
    (* Write control commands to IED *)
    (* WRITE_IED_CONTROL(device_name, 'LD0/CSWI1$CO$Pos', TRUE); *)
END_IF;
*)

(* ====== Built-in Functions Available ====== *)
(*
   READ_IED_DATA(device: STRING, ref: STRING): ANY
       - Read data from IED object reference
       - Example: READ_IED_DATA('MyIED', 'LD0/MMXU1$MX$TotW$mag')

   WRITE_IED_DATA(device: STRING, ref: STRING, value: ANY): BOOL
       - Write data to IED object reference
       - Returns TRUE on success

   WRITE_IED_CONTROL(device: STRING, ref: STRING, value: ANY): BOOL
       - Send control command to IED
       - Returns TRUE on success

   SCADA_LOG(level: STRING, message: STRING)
       - Log message to event log
       - Levels: 'INFO', 'WARNING', 'ERROR'

   GET_DEVICE_STATUS(device: STRING): BOOL
       - Check if device is connected
*)

END_PROGRAM

(* ---- PRG_GPS01GPC05UPM01FCB02.st ---- *)
(* ========================================================================
   PLC PROGRAM: PRG_GPS01GPC05UPM01FCB02
   IED: GPS01GPC05UPM01FCB02
   Device: GPS01GPC05UPM01FCB02
   Generated: 2026-02-05 10:47:40

   This program runs cyclically (default 100ms) and has access to all
   data points of the associated IEC 61850 device. Users can add custom
   logic in the designated sections below.
   ======================================================================== *)

PROGRAM PRG_GPS01GPC05UPM01FCB02
VAR
    (* ====== System Variables ====== *)
    cycle_count: UDINT := 0;           (* Increments each scan cycle *)
    first_scan: BOOL := TRUE;          (* TRUE only on first execution *)
    scan_time_ms: REAL := 0.0;         (* Last scan time in milliseconds *)

    (* ====== IED Connection Status ====== *)
    ied_connected: BOOL := FALSE;      (* TRUE when IED server is running *)
    ied_name: STRING := 'GPS01GPC05UPM01FCB02';
    device_name: STRING := 'GPS01GPC05UPM01FCB02';

    (* ====== Logical Devices ====== *)
    (* Available LDs: AnUn_ArcProtInput1, Application, BinIO, BinIO_BinaryInputs, BinIO_BinaryOutputs, CB1, CB1_Fundamental, Ds1, Ds2, Mod1, Mod1_Channel1, Mod2, Mod2_Channel1, Mod3, Mod3_Channel1, PowS, PowS_MeasPointI3ph1, PowS_MeasPointV3ph1, Rec, Rec_FaultRecorder, VI3p1, VI3p1_5051NOCgndB1, VI3p1_5051OC3phase1, VI3p1_ArcProtection1, VI3p1_Energy, VI3p1_FundSymComp, VI3p1_OperationalValues, VI3p1_ProcessMonitor, VI3p1_ExternalTrip1, VI3p1_67DirOC3phB1, VI3p1_67NDirOCgndB1, ComSupervision, ComSupervision_GOOSE *)

    (* ====== User Variables ====== *)
    (* Add your custom variables here *)
    (* Example:
    timer1: TON;
    counter: INT := 0;
    status_word: WORD;
    *)

END_VAR

(* ======================================================================
   INITIALIZATION SECTION
   Runs once on first scan. Use for setup and initialization.
   ====================================================================== *)
IF first_scan THEN
    (* Initialize user variables here *)
    cycle_count := 0;

    (* Log program start *)
    (* SCADA_LOG('INFO', CONCAT('PLC Program started: ', device_name)); *)

    first_scan := FALSE;
END_IF;

(* ======================================================================
   MAIN CYCLIC EXECUTION
   This section runs continuously every scan cycle (default 100ms).
   ====================================================================== *)

(* Increment cycle counter *)
cycle_count := cycle_count + 1;

(* ====== USER LOGIC SECTION 1: Pre-Processing ====== *)
(* Add logic that should run before main processing *)
(* Example:
IF ied_connected THEN
    (* Read IED data points *)
    (* status_word := READ_IED_DATA(device_name, 'LD0/MMXU1$MX$TotW$mag'); *)
END_IF;
*)

(* ====== USER LOGIC SECTION 2: Main Processing ====== *)
(* Add your main control logic here *)
(* Example:
IF counter > 100 THEN
    counter := 0;
    (* Perform periodic action *)
END_IF;
counter := counter + 1;
*)

(* ====== USER LOGIC SECTION 3: Post-Processing ====== *)
(* Add logic for outputs, writes, and cleanup *)
(* Example:
IF ied_connected THEN
    (* Write control commands to IED *)
    (* WRITE_IED_CONTROL(device_name, 'LD0/CSWI1$CO$Pos', TRUE); *)
END_IF;
*)

(* ====== Built-in Functions Available ====== *)
(*
   READ_IED_DATA(device: STRING, ref: STRING): ANY
       - Read data from IED object reference
       - Example: READ_IED_DATA('MyIED', 'LD0/MMXU1$MX$TotW$mag')

   WRITE_IED_DATA(device: STRING, ref: STRING, value: ANY): BOOL
       - Write data to IED object reference
       - Returns TRUE on success

   WRITE_IED_CONTROL(device: STRING, ref: STRING, value: ANY): BOOL
       - Send control command to IED
       - Returns TRUE on success

   SCADA_LOG(level: STRING, message: STRING)
       - Log message to event log
       - Levels: 'INFO', 'WARNING', 'ERROR'

   GET_DEVICE_STATUS(device: STRING): BOOL
       - Check if device is connected
*)

END_PROGRAM

(* ---- PRG_GPS01GPC05UPM01MCB01.st ---- *)
(* ========================================================================
   PLC PROGRAM: PRG_GPS01GPC05UPM01MCB01
   IED: GPS01GPC05UPM01MCB01
   Device: GPS01GPC05UPM01MCB01
   Generated: 2026-02-05 10:47:42

   This program runs cyclically (default 100ms) and has access to all
   data points of the associated IEC 61850 device. Users can add custom
   logic in the designated sections below.
   ======================================================================== *)

PROGRAM PRG_GPS01GPC05UPM01MCB01
VAR
    (* ====== System Variables ====== *)
    cycle_count: UDINT := 0;           (* Increments each scan cycle *)
    first_scan: BOOL := TRUE;          (* TRUE only on first execution *)
    scan_time_ms: REAL := 0.0;         (* Last scan time in milliseconds *)

    (* ====== IED Connection Status ====== *)
    ied_connected: BOOL := FALSE;      (* TRUE when IED server is running *)
    ied_name: STRING := 'GPS01GPC05UPM01MCB01';
    device_name: STRING := 'GPS01GPC05UPM01MCB01';

    (* ====== Logical Devices ====== *)
    (* Available LDs: AnUn_ArcProtInput1, Application, BinIO, BinIO_BinaryInputs, BinIO_BinaryOutputs, CB1, CB1_Fundamental, Ds1, Ds2, Mod1, Mod1_Channel1, Mod2, Mod2_Channel1, Mod3, Mod3_Channel1, PowS, PowS_MeasPointI3ph1, PowS_MeasPointV3ph1, Rec, Rec_FaultRecorder, VI3p1, VI3p1_5051NOCgndB1, VI3p1_5051OC3phase1, VI3p1_ArcProtection1, VI3p1_Energy, VI3p1_FundSymComp, VI3p1_OperationalValues, VI3p1_ProcessMonitor, VI3p1_ExternalTrip1, VI3p1_67DirOC3phB1, VI3p1_67NDirOCgndB1, VI3p1_ExternalTrip2, ComSupervision, ComSupervision_GOOSE *)

    (* ====== User Variables ====== *)
    (* Add your custom variables here *)
    (* Example:
    timer1: TON;
    counter: INT := 0;
    status_word: WORD;
    *)

END_VAR

(* ======================================================================
   INITIALIZATION SECTION
   Runs once on first scan. Use for setup and initialization.
   ====================================================================== *)
IF first_scan THEN
    (* Initialize user variables here *)
    cycle_count := 0;

    (* Log program start *)
    (* SCADA_LOG('INFO', CONCAT('PLC Program started: ', device_name)); *)

    first_scan := FALSE;
END_IF;

(* ======================================================================
   MAIN CYCLIC EXECUTION
   This section runs continuously every scan cycle (default 100ms).
   ====================================================================== *)

(* Increment cycle counter *)
cycle_count := cycle_count + 1;

(* ====== USER LOGIC SECTION 1: Pre-Processing ====== *)
(* Add logic that should run before main processing *)
(* Example:
IF ied_connected THEN
    (* Read IED data points *)
    (* status_word := READ_IED_DATA(device_name, 'LD0/MMXU1$MX$TotW$mag'); *)
END_IF;
*)

(* ====== USER LOGIC SECTION 2: Main Processing ====== *)
(* Add your main control logic here *)
(* Example:
IF counter > 100 THEN
    counter := 0;
    (* Perform periodic action *)
END_IF;
counter := counter + 1;
*)

(* ====== USER LOGIC SECTION 3: Post-Processing ====== *)
(* Add logic for outputs, writes, and cleanup *)
(* Example:
IF ied_connected THEN
    (* Write control commands to IED *)
    (* WRITE_IED_CONTROL(device_name, 'LD0/CSWI1$CO$Pos', TRUE); *)
END_IF;
*)

(* ====== Built-in Functions Available ====== *)
(*
   READ_IED_DATA(device: STRING, ref: STRING): ANY
       - Read data from IED object reference
       - Example: READ_IED_DATA('MyIED', 'LD0/MMXU1$MX$TotW$mag')

   WRITE_IED_DATA(device: STRING, ref: STRING, value: ANY): BOOL
       - Write data to IED object reference
       - Returns TRUE on success

   WRITE_IED_CONTROL(device: STRING, ref: STRING, value: ANY): BOOL
       - Send control command to IED
       - Returns TRUE on success

   SCADA_LOG(level: STRING, message: STRING)
       - Log message to event log
       - Levels: 'INFO', 'WARNING', 'ERROR'

   GET_DEVICE_STATUS(device: STRING): BOOL
       - Check if device is connected
*)

END_PROGRAM

(* ---- PRG_GPS01LBB01.st ---- *)
(* ========================================================================
   PLC PROGRAM: PRG_GPS01LBB01
   IED: GPS01LBB01
   Device: GPS01LBB01
   Generated: 2026-02-05 10:51:11

   This program runs cyclically (default 100ms) and has access to all
   data points of the associated IEC 61850 device. Users can add custom
   logic in the designated sections below.
   ======================================================================== *)

PROGRAM PRG_GPS01LBB01
VAR
    (* ====== System Variables ====== *)
    cycle_count: UDINT := 0;           (* Increments each scan cycle *)
    first_scan: BOOL := TRUE;          (* TRUE only on first execution *)
    scan_time_ms: REAL := 0.0;         (* Last scan time in milliseconds *)

    (* ====== IED Connection Status ====== *)
    ied_connected: BOOL := FALSE;      (* TRUE when IED server is running *)
    ied_name: STRING := 'GPS01LBB01';
    device_name: STRING := 'GPS01LBB01';

    (* ====== Logical Devices ====== *)
    (* Available LDs: AnUn_ArcProtInput1, Application, BinIO, BinIO_BinaryInputs, BinIO_BinaryOutputs, CB1, CB1_Fundamental, Ds1, Ds2, Mod1, Mod1_Channel1, Mod2, Mod2_Channel1, Mod3, Mod3_Channel1, PowS, PowS_MeasPointI3ph1, PowS_MeasPointV3ph1, Rec, Rec_FaultRecorder, VI3p1, VI3p1_5051NOCgndB1, VI3p1_5051OC3phase1, VI3p1_67DirOC3phB1, VI3p1_67NDirOCgndB1, VI3p1_ArcProtection1, VI3p1_Energy, VI3p1_FundSymComp, VI3p1_OperationalValues, VI3p1_ProcessMonitor, VI3p1_ExternalTrip1, VI3p1_ExternalTrip2, VI3p1_ExternalTrip3, ComSupervision, ComSupervision_GOOSE *)

    (* ====== User Variables ====== *)
    (* Add your custom variables here *)
    (* Example:
    timer1: TON;
    counter: INT := 0;
    status_word: WORD;
    *)

END_VAR

(* ======================================================================
   INITIALIZATION SECTION
   Runs once on first scan. Use for setup and initialization.
   ====================================================================== *)
IF first_scan THEN
    (* Initialize user variables here *)
    cycle_count := 0;

    (* Log program start *)
    (* SCADA_LOG('INFO', CONCAT('PLC Program started: ', device_name)); *)

    first_scan := FALSE;
END_IF;

(* ======================================================================
   MAIN CYCLIC EXECUTION
   This section runs continuously every scan cycle (default 100ms).
   ====================================================================== *)

(* Increment cycle counter *)
cycle_count := cycle_count + 1;

(* ====== USER LOGIC SECTION 1: Pre-Processing ====== *)
(* Add logic that should run before main processing *)
(* Example:
IF ied_connected THEN
    (* Read IED data points *)
    (* status_word := READ_IED_DATA(device_name, 'LD0/MMXU1$MX$TotW$mag'); *)
END_IF;
*)

(* ====== USER LOGIC SECTION 2: Main Processing ====== *)
(* Add your main control logic here *)
(* Example:
IF counter > 100 THEN
    counter := 0;
    (* Perform periodic action *)
END_IF;
counter := counter + 1;
*)

(* ====== USER LOGIC SECTION 3: Post-Processing ====== *)
(* Add logic for outputs, writes, and cleanup *)
(* Example:
IF ied_connected THEN
    (* Write control commands to IED *)
    (* WRITE_IED_CONTROL(device_name, 'LD0/CSWI1$CO$Pos', TRUE); *)
END_IF;
*)

(* ====== Built-in Functions Available ====== *)
(*
   READ_IED_DATA(device: STRING, ref: STRING): ANY
       - Read data from IED object reference
       - Example: READ_IED_DATA('MyIED', 'LD0/MMXU1$MX$TotW$mag')

   WRITE_IED_DATA(device: STRING, ref: STRING, value: ANY): BOOL
       - Write data to IED object reference
       - Returns TRUE on success

   WRITE_IED_CONTROL(device: STRING, ref: STRING, value: ANY): BOOL
       - Send control command to IED
       - Returns TRUE on success

   SCADA_LOG(level: STRING, message: STRING)
       - Log message to event log
       - Levels: 'INFO', 'WARNING', 'ERROR'

   GET_DEVICE_STATUS(device: STRING): BOOL
       - Check if device is connected
*)

END_PROGRAM

(* ---- PRG_GPS01MCB01.st ---- *)
(* ========================================================================
   PLC PROGRAM: PRG_GPS01MCB01
   IED: GPS01MCB01
   Device: GPS01MCB01
   Generated: 2026-02-05 10:50:26

   This program runs cyclically (default 100ms) and has access to all
   data points of the associated IEC 61850 device. Users can add custom
   logic in the designated sections below.
   ======================================================================== *)

PROGRAM PRG_GPS01MCB01
VAR
    (* ====== System Variables ====== *)
    cycle_count: UDINT := 0;           (* Increments each scan cycle *)
    first_scan: BOOL := TRUE;          (* TRUE only on first execution *)
    scan_time_ms: REAL := 0.0;         (* Last scan time in milliseconds *)

    (* ====== IED Connection Status ====== *)
    ied_connected: BOOL := FALSE;      (* TRUE when IED server is running *)
    ied_name: STRING := 'GPS01MCB01';
    device_name: STRING := 'GPS01MCB01';

    (* ====== Logical Devices ====== *)
    (* Available LDs: AnUn_ArcProtInput1, Application, BinIO, BinIO_BinaryInputs, BinIO_BinaryOutputs, CB1, CB1_Fundamental, Ds1, Ds2, Mod1, Mod1_Channel1, Mod2, Mod2_Channel1, Mod3, Mod3_Channel1, PowS, PowS_MeasPointI3ph1, PowS_MeasPointV1ph1, PowS_MeasPointV3ph1, Rec, Rec_FaultRecorder, VI1p1, VI1p1_Fundamental, VI3p1, VI3p1_5051NOCgndB1, VI3p1_5051OC3phase1, VI3p1_67DirOC3phB1, VI3p1_67NDirOCgndB1, VI3p1_ArcProtection1, VI3p1_Energy, VI3p1_FundSymComp, VI3p1_OperationalValues, VI3p1_ProcessMonitor, VI3p1_ExternalTrip1, VI3p1_ExternalTrip2, VI3p1_ExternalTrip3, ComSupervision, ComSupervision_GOOSE *)

    (* ====== User Variables ====== *)
    (* Add your custom variables here *)
    (* Example:
    timer1: TON;
    counter: INT := 0;
    status_word: WORD;
    *)

END_VAR

(* ======================================================================
   INITIALIZATION SECTION
   Runs once on first scan. Use for setup and initialization.
   ====================================================================== *)
IF first_scan THEN
    (* Initialize user variables here *)
    cycle_count := 0;

    (* Log program start *)
    (* SCADA_LOG('INFO', CONCAT('PLC Program started: ', device_name)); *)

    first_scan := FALSE;
END_IF;

(* ======================================================================
   MAIN CYCLIC EXECUTION
   This section runs continuously every scan cycle (default 100ms).
   ====================================================================== *)

(* Increment cycle counter *)
cycle_count := cycle_count + 1;

(* ====== USER LOGIC SECTION 1: Pre-Processing ====== *)
(* Add logic that should run before main processing *)
(* Example:
IF ied_connected THEN
    (* Read IED data points *)
    (* status_word := READ_IED_DATA(device_name, 'LD0/MMXU1$MX$TotW$mag'); *)
END_IF;
*)

(* ====== USER LOGIC SECTION 2: Main Processing ====== *)
(* Add your main control logic here *)
(* Example:
IF counter > 100 THEN
    counter := 0;
    (* Perform periodic action *)
END_IF;
counter := counter + 1;
*)

(* ====== USER LOGIC SECTION 3: Post-Processing ====== *)
(* Add logic for outputs, writes, and cleanup *)
(* Example:
IF ied_connected THEN
    (* Write control commands to IED *)
    (* WRITE_IED_CONTROL(device_name, 'LD0/CSWI1$CO$Pos', TRUE); *)
END_IF;
*)

(* ====== Built-in Functions Available ====== *)
(*
   READ_IED_DATA(device: STRING, ref: STRING): ANY
       - Read data from IED object reference
       - Example: READ_IED_DATA('MyIED', 'LD0/MMXU1$MX$TotW$mag')

   WRITE_IED_DATA(device: STRING, ref: STRING, value: ANY): BOOL
       - Write data to IED object reference
       - Returns TRUE on success

   WRITE_IED_CONTROL(device: STRING, ref: STRING, value: ANY): BOOL
       - Send control command to IED
       - Returns TRUE on success

   SCADA_LOG(level: STRING, message: STRING)
       - Log message to event log
       - Levels: 'INFO', 'WARNING', 'ERROR'

   GET_DEVICE_STATUS(device: STRING): BOOL
       - Check if device is connected
*)

END_PROGRAM

(* ---- PRG_GPS02ECB01.st ---- *)
(* ========================================================================
   PLC PROGRAM: PRG_GPS02ECB01
   IED: GPS02ECB01
   Device: GPS02ECB01
   Generated: 2026-02-05 10:51:32

   This program runs cyclically (default 100ms) and has access to all
   data points of the associated IEC 61850 device. Users can add custom
   logic in the designated sections below.
   ======================================================================== *)

PROGRAM PRG_GPS02ECB01
VAR
    (* ====== System Variables ====== *)
    cycle_count: UDINT := 0;           (* Increments each scan cycle *)
    first_scan: BOOL := TRUE;          (* TRUE only on first execution *)
    scan_time_ms: REAL := 0.0;         (* Last scan time in milliseconds *)

    (* ====== IED Connection Status ====== *)
    ied_connected: BOOL := FALSE;      (* TRUE when IED server is running *)
    ied_name: STRING := 'GPS02ECB01';
    device_name: STRING := 'GPS02ECB01';

    (* ====== Logical Devices ====== *)
    (* Available LDs: AnUn_ArcProtInput1, Application, BinIO, BinIO_BinaryInputs, BinIO_BinaryOutputs, CB1, CB1_Fundamental, Ds1, Ds2, Mod1, Mod1_Channel1, Mod2, Mod2_Channel1, Mod3, Mod3_Channel1, PowS, PowS_MeasPointI3ph1, PowS_MeasPointV3ph1, Rec, Rec_FaultRecorder, VI3p1, VI3p1_5051NOCgndB1, VI3p1_5051OC3phase1, VI3p1_67DirOC3phB1, VI3p1_67NDirOCgndB1, VI3p1_ArcProtection1, VI3p1_Energy, VI3p1_FundSymComp, VI3p1_OperationalValues, VI3p1_ProcessMonitor, VI3p1_ExternalTrip1, VI3p1_ExternalTrip2, PowS_MeasPointI1ph1, VI1p1, VI1p1_50N51NOC1phB1, VI1p1_Fundamental, ComSupervision, ComSupervision_GOOSE *)

    (* ====== User Variables ====== *)
    (* Add your custom variables here *)
    (* Example:
    timer1: TON;
    counter: INT := 0;
    status_word: WORD;
    *)

END_VAR

(* ======================================================================
   INITIALIZATION SECTION
   Runs once on first scan. Use for setup and initialization.
   ====================================================================== *)
IF first_scan THEN
    (* Initialize user variables here *)
    cycle_count := 0;

    (* Log program start *)
    (* SCADA_LOG('INFO', CONCAT('PLC Program started: ', device_name)); *)

    first_scan := FALSE;
END_IF;

(* ======================================================================
   MAIN CYCLIC EXECUTION
   This section runs continuously every scan cycle (default 100ms).
   ====================================================================== *)

(* Increment cycle counter *)
cycle_count := cycle_count + 1;

(* ====== USER LOGIC SECTION 1: Pre-Processing ====== *)
(* Add logic that should run before main processing *)
(* Example:
IF ied_connected THEN
    (* Read IED data points *)
    (* status_word := READ_IED_DATA(device_name, 'LD0/MMXU1$MX$TotW$mag'); *)
END_IF;
*)

(* ====== USER LOGIC SECTION 2: Main Processing ====== *)
(* Add your main control logic here *)
(* Example:
IF counter > 100 THEN
    counter := 0;
    (* Perform periodic action *)
END_IF;
counter := counter + 1;
*)

(* ====== USER LOGIC SECTION 3: Post-Processing ====== *)
(* Add logic for outputs, writes, and cleanup *)
(* Example:
IF ied_connected THEN
    (* Write control commands to IED *)
    (* WRITE_IED_CONTROL(device_name, 'LD0/CSWI1$CO$Pos', TRUE); *)
END_IF;
*)

(* ====== Built-in Functions Available ====== *)
(*
   READ_IED_DATA(device: STRING, ref: STRING): ANY
       - Read data from IED object reference
       - Example: READ_IED_DATA('MyIED', 'LD0/MMXU1$MX$TotW$mag')

   WRITE_IED_DATA(device: STRING, ref: STRING, value: ANY): BOOL
       - Write data to IED object reference
       - Returns TRUE on success

   WRITE_IED_CONTROL(device: STRING, ref: STRING, value: ANY): BOOL
       - Send control command to IED
       - Returns TRUE on success

   SCADA_LOG(level: STRING, message: STRING)
       - Log message to event log
       - Levels: 'INFO', 'WARNING', 'ERROR'

   GET_DEVICE_STATUS(device: STRING): BOOL
       - Check if device is connected
*)

END_PROGRAM

(* ---- PRG_GPS02FCB01.st ---- *)
(* ========================================================================
   PLC PROGRAM: PRG_GPS02FCB01
   IED: GPS02FCB01
   Device: GPS02FCB01
   Generated: 2026-02-05 10:51:43

   This program runs cyclically (default 100ms) and has access to all
   data points of the associated IEC 61850 device. Users can add custom
   logic in the designated sections below.
   ======================================================================== *)

PROGRAM PRG_GPS02FCB01
VAR
    (* ====== System Variables ====== *)
    cycle_count: UDINT := 0;           (* Increments each scan cycle *)
    first_scan: BOOL := TRUE;          (* TRUE only on first execution *)
    scan_time_ms: REAL := 0.0;         (* Last scan time in milliseconds *)

    (* ====== IED Connection Status ====== *)
    ied_connected: BOOL := FALSE;      (* TRUE when IED server is running *)
    ied_name: STRING := 'GPS02FCB01';
    device_name: STRING := 'GPS02FCB01';

    (* ====== Logical Devices ====== *)
    (* Available LDs: AnUn_ArcProtInput1, Application, BinIO, BinIO_BinaryInputs, BinIO_BinaryOutputs, CB1, CB1_Fundamental, Ds1, Ds2, Mod1, Mod1_Channel1, Mod2, Mod2_Channel1, Mod3, Mod3_Channel1, PowS, PowS_MeasPointI3ph1, PowS_MeasPointV1ph1, PowS_MeasPointV3ph1, Rec, Rec_FaultRecorder, VI1p1, VI1p1_Fundamental, VI3p1, VI3p1_5051NOCgndB1, VI3p1_5051OC3phase1, VI3p1_67DirOC3phB1, VI3p1_67NDirOCgndB1, VI3p1_ArcProtection1, VI3p1_Energy, VI3p1_FundSymComp, VI3p1_OperationalValues, VI3p1_ProcessMonitor, VI3p1_ExternalTrip1, VI3p1_ExternalTrip2, ComSupervision, ComSupervision_GOOSE *)

    (* ====== User Variables ====== *)
    (* Add your custom variables here *)
    (* Example:
    timer1: TON;
    counter: INT := 0;
    status_word: WORD;
    *)

END_VAR

(* ======================================================================
   INITIALIZATION SECTION
   Runs once on first scan. Use for setup and initialization.
   ====================================================================== *)
IF first_scan THEN
    (* Initialize user variables here *)
    cycle_count := 0;

    (* Log program start *)
    (* SCADA_LOG('INFO', CONCAT('PLC Program started: ', device_name)); *)

    first_scan := FALSE;
END_IF;

(* ======================================================================
   MAIN CYCLIC EXECUTION
   This section runs continuously every scan cycle (default 100ms).
   ====================================================================== *)

(* Increment cycle counter *)
cycle_count := cycle_count + 1;

(* ====== USER LOGIC SECTION 1: Pre-Processing ====== *)
(* Add logic that should run before main processing *)
(* Example:
IF ied_connected THEN
    (* Read IED data points *)
    (* status_word := READ_IED_DATA(device_name, 'LD0/MMXU1$MX$TotW$mag'); *)
END_IF;
*)

(* ====== USER LOGIC SECTION 2: Main Processing ====== *)
(* Add your main control logic here *)
(* Example:
IF counter > 100 THEN
    counter := 0;
    (* Perform periodic action *)
END_IF;
counter := counter + 1;
*)

(* ====== USER LOGIC SECTION 3: Post-Processing ====== *)
(* Add logic for outputs, writes, and cleanup *)
(* Example:
IF ied_connected THEN
    (* Write control commands to IED *)
    (* WRITE_IED_CONTROL(device_name, 'LD0/CSWI1$CO$Pos', TRUE); *)
END_IF;
*)

(* ====== Built-in Functions Available ====== *)
(*
   READ_IED_DATA(device: STRING, ref: STRING): ANY
       - Read data from IED object reference
       - Example: READ_IED_DATA('MyIED', 'LD0/MMXU1$MX$TotW$mag')

   WRITE_IED_DATA(device: STRING, ref: STRING, value: ANY): BOOL
       - Write data to IED object reference
       - Returns TRUE on success

   WRITE_IED_CONTROL(device: STRING, ref: STRING, value: ANY): BOOL
       - Send control command to IED
       - Returns TRUE on success

   SCADA_LOG(level: STRING, message: STRING)
       - Log message to event log
       - Levels: 'INFO', 'WARNING', 'ERROR'

   GET_DEVICE_STATUS(device: STRING): BOOL
       - Check if device is connected
*)

END_PROGRAM

(* ---- PRG_GPS02FCB02.st ---- *)
(* ========================================================================
   PLC PROGRAM: PRG_GPS02FCB02
   IED: GPS02FCB02
   Device: GPS02FCB02
   Generated: 2026-02-05 10:51:41

   This program runs cyclically (default 100ms) and has access to all
   data points of the associated IEC 61850 device. Users can add custom
   logic in the designated sections below.
   ======================================================================== *)

PROGRAM PRG_GPS02FCB02
VAR
    (* ====== System Variables ====== *)
    cycle_count: UDINT := 0;           (* Increments each scan cycle *)
    first_scan: BOOL := TRUE;          (* TRUE only on first execution *)
    scan_time_ms: REAL := 0.0;         (* Last scan time in milliseconds *)

    (* ====== IED Connection Status ====== *)
    ied_connected: BOOL := FALSE;      (* TRUE when IED server is running *)
    ied_name: STRING := 'GPS02FCB02';
    device_name: STRING := 'GPS02FCB02';

    (* ====== Logical Devices ====== *)
    (* Available LDs: AnUn_ArcProtInput1, Application, BinIO, BinIO_BinaryInputs, BinIO_BinaryOutputs, CB1, CB1_Fundamental, Ds1, Ds2, Mod1, Mod1_Channel1, Mod2, Mod2_Channel1, Mod3, Mod3_Channel1, PowS, PowS_MeasPointI3ph1, PowS_MeasPointV1ph1, PowS_MeasPointV3ph1, Rec, Rec_FaultRecorder, VI1p1, VI1p1_Fundamental, VI3p1, VI3p1_5051NOCgndB1, VI3p1_5051OC3phase1, VI3p1_67DirOC3phB1, VI3p1_67NDirOCgndB1, VI3p1_ArcProtection1, VI3p1_Energy, VI3p1_FundSymComp, VI3p1_OperationalValues, VI3p1_ProcessMonitor, VI3p1_ExternalTrip1, VI3p1_ExternalTrip2, ComSupervision, ComSupervision_GOOSE *)

    (* ====== User Variables ====== *)
    (* Add your custom variables here *)
    (* Example:
    timer1: TON;
    counter: INT := 0;
    status_word: WORD;
    *)

END_VAR

(* ======================================================================
   INITIALIZATION SECTION
   Runs once on first scan. Use for setup and initialization.
   ====================================================================== *)
IF first_scan THEN
    (* Initialize user variables here *)
    cycle_count := 0;

    (* Log program start *)
    (* SCADA_LOG('INFO', CONCAT('PLC Program started: ', device_name)); *)

    first_scan := FALSE;
END_IF;

(* ======================================================================
   MAIN CYCLIC EXECUTION
   This section runs continuously every scan cycle (default 100ms).
   ====================================================================== *)

(* Increment cycle counter *)
cycle_count := cycle_count + 1;

(* ====== USER LOGIC SECTION 1: Pre-Processing ====== *)
(* Add logic that should run before main processing *)
(* Example:
IF ied_connected THEN
    (* Read IED data points *)
    (* status_word := READ_IED_DATA(device_name, 'LD0/MMXU1$MX$TotW$mag'); *)
END_IF;
*)

(* ====== USER LOGIC SECTION 2: Main Processing ====== *)
(* Add your main control logic here *)
(* Example:
IF counter > 100 THEN
    counter := 0;
    (* Perform periodic action *)
END_IF;
counter := counter + 1;
*)

(* ====== USER LOGIC SECTION 3: Post-Processing ====== *)
(* Add logic for outputs, writes, and cleanup *)
(* Example:
IF ied_connected THEN
    (* Write control commands to IED *)
    (* WRITE_IED_CONTROL(device_name, 'LD0/CSWI1$CO$Pos', TRUE); *)
END_IF;
*)

(* ====== Built-in Functions Available ====== *)
(*
   READ_IED_DATA(device: STRING, ref: STRING): ANY
       - Read data from IED object reference
       - Example: READ_IED_DATA('MyIED', 'LD0/MMXU1$MX$TotW$mag')

   WRITE_IED_DATA(device: STRING, ref: STRING, value: ANY): BOOL
       - Write data to IED object reference
       - Returns TRUE on success

   WRITE_IED_CONTROL(device: STRING, ref: STRING, value: ANY): BOOL
       - Send control command to IED
       - Returns TRUE on success

   SCADA_LOG(level: STRING, message: STRING)
       - Log message to event log
       - Levels: 'INFO', 'WARNING', 'ERROR'

   GET_DEVICE_STATUS(device: STRING): BOOL
       - Check if device is connected
*)

END_PROGRAM

(* ---- PRG_GPS02FCB03.st ---- *)
(* ========================================================================
   PLC PROGRAM: PRG_GPS02FCB03
   IED: GPS02FCB03
   Device: GPS02FCB03
   Generated: 2026-02-05 10:52:29

   This program runs cyclically (default 100ms) and has access to all
   data points of the associated IEC 61850 device. Users can add custom
   logic in the designated sections below.
   ======================================================================== *)

PROGRAM PRG_GPS02FCB03
VAR
    (* ====== System Variables ====== *)
    cycle_count: UDINT := 0;           (* Increments each scan cycle *)
    first_scan: BOOL := TRUE;          (* TRUE only on first execution *)
    scan_time_ms: REAL := 0.0;         (* Last scan time in milliseconds *)

    (* ====== IED Connection Status ====== *)
    ied_connected: BOOL := FALSE;      (* TRUE when IED server is running *)
    ied_name: STRING := 'GPS02FCB03';
    device_name: STRING := 'GPS02FCB03';

    (* ====== Logical Devices ====== *)
    (* Available LDs: AnUn_ArcProtInput1, Application, BinIO, BinIO_BinaryInputs, BinIO_BinaryOutputs, CB1, CB1_Fundamental, Ds1, Ds2, Mod1, Mod1_Channel1, Mod2, Mod2_Channel1, Mod3, Mod3_Channel1, PowS, PowS_MeasPointI3ph1, PowS_MeasPointV1ph1, PowS_MeasPointV3ph1, Rec, Rec_FaultRecorder, VI1p1, VI1p1_Fundamental, VI3p1, VI3p1_5051NOCgndB1, VI3p1_5051OC3phase1, VI3p1_67DirOC3phB1, VI3p1_67NDirOCgndB1, VI3p1_ArcProtection1, VI3p1_Energy, VI3p1_FundSymComp, VI3p1_OperationalValues, VI3p1_ProcessMonitor, VI3p1_ExternalTrip1, VI3p1_ExternalTrip2, ComSupervision, ComSupervision_GOOSE *)

    (* ====== User Variables ====== *)
    (* Add your custom variables here *)
    (* Example:
    timer1: TON;
    counter: INT := 0;
    status_word: WORD;
    *)

END_VAR

(* ======================================================================
   INITIALIZATION SECTION
   Runs once on first scan. Use for setup and initialization.
   ====================================================================== *)
IF first_scan THEN
    (* Initialize user variables here *)
    cycle_count := 0;

    (* Log program start *)
    (* SCADA_LOG('INFO', CONCAT('PLC Program started: ', device_name)); *)

    first_scan := FALSE;
END_IF;

(* ======================================================================
   MAIN CYCLIC EXECUTION
   This section runs continuously every scan cycle (default 100ms).
   ====================================================================== *)

(* Increment cycle counter *)
cycle_count := cycle_count + 1;

(* ====== USER LOGIC SECTION 1: Pre-Processing ====== *)
(* Add logic that should run before main processing *)
(* Example:
IF ied_connected THEN
    (* Read IED data points *)
    (* status_word := READ_IED_DATA(device_name, 'LD0/MMXU1$MX$TotW$mag'); *)
END_IF;
*)

(* ====== USER LOGIC SECTION 2: Main Processing ====== *)
(* Add your main control logic here *)
(* Example:
IF counter > 100 THEN
    counter := 0;
    (* Perform periodic action *)
END_IF;
counter := counter + 1;
*)

(* ====== USER LOGIC SECTION 3: Post-Processing ====== *)
(* Add logic for outputs, writes, and cleanup *)
(* Example:
IF ied_connected THEN
    (* Write control commands to IED *)
    (* WRITE_IED_CONTROL(device_name, 'LD0/CSWI1$CO$Pos', TRUE); *)
END_IF;
*)

(* ====== Built-in Functions Available ====== *)
(*
   READ_IED_DATA(device: STRING, ref: STRING): ANY
       - Read data from IED object reference
       - Example: READ_IED_DATA('MyIED', 'LD0/MMXU1$MX$TotW$mag')

   WRITE_IED_DATA(device: STRING, ref: STRING, value: ANY): BOOL
       - Write data to IED object reference
       - Returns TRUE on success

   WRITE_IED_CONTROL(device: STRING, ref: STRING, value: ANY): BOOL
       - Send control command to IED
       - Returns TRUE on success

   SCADA_LOG(level: STRING, message: STRING)
       - Log message to event log
       - Levels: 'INFO', 'WARNING', 'ERROR'

   GET_DEVICE_STATUS(device: STRING): BOOL
       - Check if device is connected
*)

END_PROGRAM

(* ---- PRG_GPS02FCB04.st ---- *)
(* ========================================================================
   PLC PROGRAM: PRG_GPS02FCB04
   IED: GPS02FCB04
   Device: GPS02FCB04
   Generated: 2026-02-05 10:51:27

   This program runs cyclically (default 100ms) and has access to all
   data points of the associated IEC 61850 device. Users can add custom
   logic in the designated sections below.
   ======================================================================== *)

PROGRAM PRG_GPS02FCB04
VAR
    (* ====== System Variables ====== *)
    cycle_count: UDINT := 0;           (* Increments each scan cycle *)
    first_scan: BOOL := TRUE;          (* TRUE only on first execution *)
    scan_time_ms: REAL := 0.0;         (* Last scan time in milliseconds *)

    (* ====== IED Connection Status ====== *)
    ied_connected: BOOL := FALSE;      (* TRUE when IED server is running *)
    ied_name: STRING := 'GPS02FCB04';
    device_name: STRING := 'GPS02FCB04';

    (* ====== Logical Devices ====== *)
    (* Available LDs: AnUn_ArcProtInput1, Application, BinIO, BinIO_BinaryInputs, BinIO_BinaryOutputs, CB1, CB1_Fundamental, Ds1, Ds2, Mod1, Mod1_Channel1, Mod2, Mod2_Channel1, Mod3, Mod3_Channel1, PowS, PowS_MeasPointI3ph1, PowS_MeasPointV1ph1, PowS_MeasPointV3ph1, Rec, Rec_FaultRecorder, VI1p1, VI1p1_Fundamental, VI3p1, VI3p1_5051NOCgndB1, VI3p1_5051OC3phase1, VI3p1_67DirOC3phB1, VI3p1_67NDirOCgndB1, VI3p1_ArcProtection1, VI3p1_Energy, VI3p1_FundSymComp, VI3p1_OperationalValues, VI3p1_ProcessMonitor, VI3p1_ExternalTrip1, VI3p1_ExternalTrip2, VI3p1_ExternalTrip3, ComSupervision, ComSupervision_GOOSE *)

    (* ====== User Variables ====== *)
    (* Add your custom variables here *)
    (* Example:
    timer1: TON;
    counter: INT := 0;
    status_word: WORD;
    *)

END_VAR

(* ======================================================================
   INITIALIZATION SECTION
   Runs once on first scan. Use for setup and initialization.
   ====================================================================== *)
IF first_scan THEN
    (* Initialize user variables here *)
    cycle_count := 0;

    (* Log program start *)
    (* SCADA_LOG('INFO', CONCAT('PLC Program started: ', device_name)); *)

    first_scan := FALSE;
END_IF;

(* ======================================================================
   MAIN CYCLIC EXECUTION
   This section runs continuously every scan cycle (default 100ms).
   ====================================================================== *)

(* Increment cycle counter *)
cycle_count := cycle_count + 1;

(* ====== USER LOGIC SECTION 1: Pre-Processing ====== *)
(* Add logic that should run before main processing *)
(* Example:
IF ied_connected THEN
    (* Read IED data points *)
    (* status_word := READ_IED_DATA(device_name, 'LD0/MMXU1$MX$TotW$mag'); *)
END_IF;
*)

(* ====== USER LOGIC SECTION 2: Main Processing ====== *)
(* Add your main control logic here *)
(* Example:
IF counter > 100 THEN
    counter := 0;
    (* Perform periodic action *)
END_IF;
counter := counter + 1;
*)

(* ====== USER LOGIC SECTION 3: Post-Processing ====== *)
(* Add logic for outputs, writes, and cleanup *)
(* Example:
IF ied_connected THEN
    (* Write control commands to IED *)
    (* WRITE_IED_CONTROL(device_name, 'LD0/CSWI1$CO$Pos', TRUE); *)
END_IF;
*)

(* ====== Built-in Functions Available ====== *)
(*
   READ_IED_DATA(device: STRING, ref: STRING): ANY
       - Read data from IED object reference
       - Example: READ_IED_DATA('MyIED', 'LD0/MMXU1$MX$TotW$mag')

   WRITE_IED_DATA(device: STRING, ref: STRING, value: ANY): BOOL
       - Write data to IED object reference
       - Returns TRUE on success

   WRITE_IED_CONTROL(device: STRING, ref: STRING, value: ANY): BOOL
       - Send control command to IED
       - Returns TRUE on success

   SCADA_LOG(level: STRING, message: STRING)
       - Log message to event log
       - Levels: 'INFO', 'WARNING', 'ERROR'

   GET_DEVICE_STATUS(device: STRING): BOOL
       - Check if device is connected
*)

END_PROGRAM

(* ---- PRG_GPS02FCB05.st ---- *)
(* ========================================================================
   PLC PROGRAM: PRG_GPS02FCB05
   IED: GPS02FCB05
   Device: GPS02FCB05
   Generated: 2026-02-05 10:52:27

   This program runs cyclically (default 100ms) and has access to all
   data points of the associated IEC 61850 device. Users can add custom
   logic in the designated sections below.
   ======================================================================== *)

PROGRAM PRG_GPS02FCB05
VAR
    (* ====== System Variables ====== *)
    cycle_count: UDINT := 0;           (* Increments each scan cycle *)
    first_scan: BOOL := TRUE;          (* TRUE only on first execution *)
    scan_time_ms: REAL := 0.0;         (* Last scan time in milliseconds *)

    (* ====== IED Connection Status ====== *)
    ied_connected: BOOL := FALSE;      (* TRUE when IED server is running *)
    ied_name: STRING := 'GPS02FCB05';
    device_name: STRING := 'GPS02FCB05';

    (* ====== Logical Devices ====== *)
    (* Available LDs: AnUn_ArcProtInput1, Application, BinIO, BinIO_BinaryInputs, BinIO_BinaryOutputs, CB1, CB1_Fundamental, Ds1, Ds2, Mod1, Mod1_Channel1, Mod2, Mod2_Channel1, Mod3, Mod3_Channel1, PowS, PowS_MeasPointI3ph1, PowS_MeasPointV1ph1, PowS_MeasPointV3ph1, Rec, Rec_FaultRecorder, VI1p1, VI1p1_Fundamental, VI3p1, VI3p1_5051NOCgndB1, VI3p1_5051OC3phase1, VI3p1_67DirOC3phB1, VI3p1_67NDirOCgndB1, VI3p1_ArcProtection1, VI3p1_Energy, VI3p1_FundSymComp, VI3p1_OperationalValues, VI3p1_ProcessMonitor, VI3p1_ExternalTrip1, VI3p1_ExternalTrip2, ComSupervision, ComSupervision_GOOSE *)

    (* ====== User Variables ====== *)
    (* Add your custom variables here *)
    (* Example:
    timer1: TON;
    counter: INT := 0;
    status_word: WORD;
    *)

END_VAR

(* ======================================================================
   INITIALIZATION SECTION
   Runs once on first scan. Use for setup and initialization.
   ====================================================================== *)
IF first_scan THEN
    (* Initialize user variables here *)
    cycle_count := 0;

    (* Log program start *)
    (* SCADA_LOG('INFO', CONCAT('PLC Program started: ', device_name)); *)

    first_scan := FALSE;
END_IF;

(* ======================================================================
   MAIN CYCLIC EXECUTION
   This section runs continuously every scan cycle (default 100ms).
   ====================================================================== *)

(* Increment cycle counter *)
cycle_count := cycle_count + 1;

(* ====== USER LOGIC SECTION 1: Pre-Processing ====== *)
(* Add logic that should run before main processing *)
(* Example:
IF ied_connected THEN
    (* Read IED data points *)
    (* status_word := READ_IED_DATA(device_name, 'LD0/MMXU1$MX$TotW$mag'); *)
END_IF;
*)

(* ====== USER LOGIC SECTION 2: Main Processing ====== *)
(* Add your main control logic here *)
(* Example:
IF counter > 100 THEN
    counter := 0;
    (* Perform periodic action *)
END_IF;
counter := counter + 1;
*)

(* ====== USER LOGIC SECTION 3: Post-Processing ====== *)
(* Add logic for outputs, writes, and cleanup *)
(* Example:
IF ied_connected THEN
    (* Write control commands to IED *)
    (* WRITE_IED_CONTROL(device_name, 'LD0/CSWI1$CO$Pos', TRUE); *)
END_IF;
*)

(* ====== Built-in Functions Available ====== *)
(*
   READ_IED_DATA(device: STRING, ref: STRING): ANY
       - Read data from IED object reference
       - Example: READ_IED_DATA('MyIED', 'LD0/MMXU1$MX$TotW$mag')

   WRITE_IED_DATA(device: STRING, ref: STRING, value: ANY): BOOL
       - Write data to IED object reference
       - Returns TRUE on success

   WRITE_IED_CONTROL(device: STRING, ref: STRING, value: ANY): BOOL
       - Send control command to IED
       - Returns TRUE on success

   SCADA_LOG(level: STRING, message: STRING)
       - Log message to event log
       - Levels: 'INFO', 'WARNING', 'ERROR'

   GET_DEVICE_STATUS(device: STRING): BOOL
       - Check if device is connected
*)

END_PROGRAM

(* ---- PRG_GPS02GCB01.st ---- *)
(* ========================================================================
   PLC PROGRAM: PRG_GPS02GCB01
   IED: GPS02GCB01
   Device: GPS02GCB01
   Generated: 2026-02-05 10:52:26

   This program runs cyclically (default 100ms) and has access to all
   data points of the associated IEC 61850 device. Users can add custom
   logic in the designated sections below.
   ======================================================================== *)

PROGRAM PRG_GPS02GCB01
VAR
    (* ====== System Variables ====== *)
    cycle_count: UDINT := 0;           (* Increments each scan cycle *)
    first_scan: BOOL := TRUE;          (* TRUE only on first execution *)
    scan_time_ms: REAL := 0.0;         (* Last scan time in milliseconds *)

    (* ====== IED Connection Status ====== *)
    ied_connected: BOOL := FALSE;      (* TRUE when IED server is running *)
    ied_name: STRING := 'GPS02GCB01';
    device_name: STRING := 'GPS02GCB01';

    (* ====== Logical Devices ====== *)
    (* Available LDs: AnUn_ArcProtInput1, Application, BinIO, BinIO_BinaryInputs, BinIO_BinaryOutputs, CB1, CB1_25Synchronization, CB1_Fundamental, Ds1, Ds2, Mod1, Mod1_Channel1, Mod2, Mod2_Channel1, Mod3, Mod3_Channel1, PowS, PowS_MeasPointI3ph1, PowS_MeasPointV1ph1, PowS_MeasPointV3ph1, Rec, Rec_FaultRecorder, VI1p1, VI1p1_Fundamental, VI3p1, VI3p1_5051NOCgndB1, VI3p1_5051OC3phase1, VI3p1_67DirOC3phB1, VI3p1_67NDirOCgndB1, VI3p1_ArcProtection1, VI3p1_Energy, VI3p1_FundSymComp, VI3p1_OperationalValues, VI3p1_ProcessMonitor, VI3p1_ExternalTrip1, VI3p1_ExternalTrip2, ComSupervision, ComSupervision_GOOSE *)

    (* ====== User Variables ====== *)
    (* Add your custom variables here *)
    (* Example:
    timer1: TON;
    counter: INT := 0;
    status_word: WORD;
    *)

END_VAR

(* ======================================================================
   INITIALIZATION SECTION
   Runs once on first scan. Use for setup and initialization.
   ====================================================================== *)
IF first_scan THEN
    (* Initialize user variables here *)
    cycle_count := 0;

    (* Log program start *)
    (* SCADA_LOG('INFO', CONCAT('PLC Program started: ', device_name)); *)

    first_scan := FALSE;
END_IF;

(* ======================================================================
   MAIN CYCLIC EXECUTION
   This section runs continuously every scan cycle (default 100ms).
   ====================================================================== *)

(* Increment cycle counter *)
cycle_count := cycle_count + 1;

(* ====== USER LOGIC SECTION 1: Pre-Processing ====== *)
(* Add logic that should run before main processing *)
(* Example:
IF ied_connected THEN
    (* Read IED data points *)
    (* status_word := READ_IED_DATA(device_name, 'LD0/MMXU1$MX$TotW$mag'); *)
END_IF;
*)

(* ====== USER LOGIC SECTION 2: Main Processing ====== *)
(* Add your main control logic here *)
(* Example:
IF counter > 100 THEN
    counter := 0;
    (* Perform periodic action *)
END_IF;
counter := counter + 1;
*)

(* ====== USER LOGIC SECTION 3: Post-Processing ====== *)
(* Add logic for outputs, writes, and cleanup *)
(* Example:
IF ied_connected THEN
    (* Write control commands to IED *)
    (* WRITE_IED_CONTROL(device_name, 'LD0/CSWI1$CO$Pos', TRUE); *)
END_IF;
*)

(* ====== Built-in Functions Available ====== *)
(*
   READ_IED_DATA(device: STRING, ref: STRING): ANY
       - Read data from IED object reference
       - Example: READ_IED_DATA('MyIED', 'LD0/MMXU1$MX$TotW$mag')

   WRITE_IED_DATA(device: STRING, ref: STRING, value: ANY): BOOL
       - Write data to IED object reference
       - Returns TRUE on success

   WRITE_IED_CONTROL(device: STRING, ref: STRING, value: ANY): BOOL
       - Send control command to IED
       - Returns TRUE on success

   SCADA_LOG(level: STRING, message: STRING)
       - Log message to event log
       - Levels: 'INFO', 'WARNING', 'ERROR'

   GET_DEVICE_STATUS(device: STRING): BOOL
       - Check if device is connected
*)

END_PROGRAM

(* ---- PRG_GPS02GCB02.st ---- *)
(* ========================================================================
   PLC PROGRAM: PRG_GPS02GCB02
   IED: GPS02GCB02
   Device: GPS02GCB02
   Generated: 2026-02-05 10:52:14

   This program runs cyclically (default 100ms) and has access to all
   data points of the associated IEC 61850 device. Users can add custom
   logic in the designated sections below.
   ======================================================================== *)

PROGRAM PRG_GPS02GCB02
VAR
    (* ====== System Variables ====== *)
    cycle_count: UDINT := 0;           (* Increments each scan cycle *)
    first_scan: BOOL := TRUE;          (* TRUE only on first execution *)
    scan_time_ms: REAL := 0.0;         (* Last scan time in milliseconds *)

    (* ====== IED Connection Status ====== *)
    ied_connected: BOOL := FALSE;      (* TRUE when IED server is running *)
    ied_name: STRING := 'GPS02GCB02';
    device_name: STRING := 'GPS02GCB02';

    (* ====== Logical Devices ====== *)
    (* Available LDs: AnUn_ArcProtInput1, Application, BinIO, BinIO_BinaryInputs, BinIO_BinaryOutputs, CB1, CB1_25Synchronization, CB1_Fundamental, Ds1, Ds2, Mod1, Mod1_Channel1, Mod2, Mod2_Channel1, Mod3, Mod3_Channel1, PowS, PowS_MeasPointI3ph1, PowS_MeasPointV1ph1, PowS_MeasPointV3ph1, Rec, Rec_FaultRecorder, VI1p1, VI1p1_Fundamental, VI3p1, VI3p1_5051NOCgndB1, VI3p1_5051OC3phase1, VI3p1_67DirOC3phB1, VI3p1_67NDirOCgndB1, VI3p1_ArcProtection1, VI3p1_Energy, VI3p1_FundSymComp, VI3p1_OperationalValues, VI3p1_ProcessMonitor, VI3p1_ExternalTrip1, VI3p1_ExternalTrip2, ComSupervision, ComSupervision_GOOSE *)

    (* ====== User Variables ====== *)
    (* Add your custom variables here *)
    (* Example:
    timer1: TON;
    counter: INT := 0;
    status_word: WORD;
    *)

END_VAR

(* ======================================================================
   INITIALIZATION SECTION
   Runs once on first scan. Use for setup and initialization.
   ====================================================================== *)
IF first_scan THEN
    (* Initialize user variables here *)
    cycle_count := 0;

    (* Log program start *)
    (* SCADA_LOG('INFO', CONCAT('PLC Program started: ', device_name)); *)

    first_scan := FALSE;
END_IF;

(* ======================================================================
   MAIN CYCLIC EXECUTION
   This section runs continuously every scan cycle (default 100ms).
   ====================================================================== *)

(* Increment cycle counter *)
cycle_count := cycle_count + 1;

(* ====== USER LOGIC SECTION 1: Pre-Processing ====== *)
(* Add logic that should run before main processing *)
(* Example:
IF ied_connected THEN
    (* Read IED data points *)
    (* status_word := READ_IED_DATA(device_name, 'LD0/MMXU1$MX$TotW$mag'); *)
END_IF;
*)

(* ====== USER LOGIC SECTION 2: Main Processing ====== *)
(* Add your main control logic here *)
(* Example:
IF counter > 100 THEN
    counter := 0;
    (* Perform periodic action *)
END_IF;
counter := counter + 1;
*)

(* ====== USER LOGIC SECTION 3: Post-Processing ====== *)
(* Add logic for outputs, writes, and cleanup *)
(* Example:
IF ied_connected THEN
    (* Write control commands to IED *)
    (* WRITE_IED_CONTROL(device_name, 'LD0/CSWI1$CO$Pos', TRUE); *)
END_IF;
*)

(* ====== Built-in Functions Available ====== *)
(*
   READ_IED_DATA(device: STRING, ref: STRING): ANY
       - Read data from IED object reference
       - Example: READ_IED_DATA('MyIED', 'LD0/MMXU1$MX$TotW$mag')

   WRITE_IED_DATA(device: STRING, ref: STRING, value: ANY): BOOL
       - Write data to IED object reference
       - Returns TRUE on success

   WRITE_IED_CONTROL(device: STRING, ref: STRING, value: ANY): BOOL
       - Send control command to IED
       - Returns TRUE on success

   SCADA_LOG(level: STRING, message: STRING)
       - Log message to event log
       - Levels: 'INFO', 'WARNING', 'ERROR'

   GET_DEVICE_STATUS(device: STRING): BOOL
       - Check if device is connected
*)

END_PROGRAM

(* ---- PRG_GPS02GCB03.st ---- *)
(* ========================================================================
   PLC PROGRAM: PRG_GPS02GCB03
   IED: GPS02GCB03
   Device: GPS02GCB03
   Generated: 2026-02-05 10:52:10

   This program runs cyclically (default 100ms) and has access to all
   data points of the associated IEC 61850 device. Users can add custom
   logic in the designated sections below.
   ======================================================================== *)

PROGRAM PRG_GPS02GCB03
VAR
    (* ====== System Variables ====== *)
    cycle_count: UDINT := 0;           (* Increments each scan cycle *)
    first_scan: BOOL := TRUE;          (* TRUE only on first execution *)
    scan_time_ms: REAL := 0.0;         (* Last scan time in milliseconds *)

    (* ====== IED Connection Status ====== *)
    ied_connected: BOOL := FALSE;      (* TRUE when IED server is running *)
    ied_name: STRING := 'GPS02GCB03';
    device_name: STRING := 'GPS02GCB03';

    (* ====== Logical Devices ====== *)
    (* Available LDs: AnUn_ArcProtInput1, Application, BinIO, BinIO_BinaryInputs, BinIO_BinaryOutputs, CB1, CB1_25Synchronization, CB1_Fundamental, Ds1, Ds2, Mod1, Mod1_Channel1, Mod2, Mod2_Channel1, Mod3, Mod3_Channel1, PowS, PowS_MeasPointI3ph1, PowS_MeasPointV1ph1, PowS_MeasPointV3ph1, Rec, Rec_FaultRecorder, VI1p1, VI1p1_Fundamental, VI3p1, VI3p1_5051NOCgndB1, VI3p1_5051OC3phase1, VI3p1_67DirOC3phB1, VI3p1_67NDirOCgndB1, VI3p1_ArcProtection1, VI3p1_Energy, VI3p1_FundSymComp, VI3p1_OperationalValues, VI3p1_ProcessMonitor, VI3p1_ExternalTrip1, VI3p1_ExternalTrip2, ComSupervision, ComSupervision_GOOSE *)

    (* ====== User Variables ====== *)
    (* Add your custom variables here *)
    (* Example:
    timer1: TON;
    counter: INT := 0;
    status_word: WORD;
    *)

END_VAR

(* ======================================================================
   INITIALIZATION SECTION
   Runs once on first scan. Use for setup and initialization.
   ====================================================================== *)
IF first_scan THEN
    (* Initialize user variables here *)
    cycle_count := 0;

    (* Log program start *)
    (* SCADA_LOG('INFO', CONCAT('PLC Program started: ', device_name)); *)

    first_scan := FALSE;
END_IF;

(* ======================================================================
   MAIN CYCLIC EXECUTION
   This section runs continuously every scan cycle (default 100ms).
   ====================================================================== *)

(* Increment cycle counter *)
cycle_count := cycle_count + 1;

(* ====== USER LOGIC SECTION 1: Pre-Processing ====== *)
(* Add logic that should run before main processing *)
(* Example:
IF ied_connected THEN
    (* Read IED data points *)
    (* status_word := READ_IED_DATA(device_name, 'LD0/MMXU1$MX$TotW$mag'); *)
END_IF;
*)

(* ====== USER LOGIC SECTION 2: Main Processing ====== *)
(* Add your main control logic here *)
(* Example:
IF counter > 100 THEN
    counter := 0;
    (* Perform periodic action *)
END_IF;
counter := counter + 1;
*)

(* ====== USER LOGIC SECTION 3: Post-Processing ====== *)
(* Add logic for outputs, writes, and cleanup *)
(* Example:
IF ied_connected THEN
    (* Write control commands to IED *)
    (* WRITE_IED_CONTROL(device_name, 'LD0/CSWI1$CO$Pos', TRUE); *)
END_IF;
*)

(* ====== Built-in Functions Available ====== *)
(*
   READ_IED_DATA(device: STRING, ref: STRING): ANY
       - Read data from IED object reference
       - Example: READ_IED_DATA('MyIED', 'LD0/MMXU1$MX$TotW$mag')

   WRITE_IED_DATA(device: STRING, ref: STRING, value: ANY): BOOL
       - Write data to IED object reference
       - Returns TRUE on success

   WRITE_IED_CONTROL(device: STRING, ref: STRING, value: ANY): BOOL
       - Send control command to IED
       - Returns TRUE on success

   SCADA_LOG(level: STRING, message: STRING)
       - Log message to event log
       - Levels: 'INFO', 'WARNING', 'ERROR'

   GET_DEVICE_STATUS(device: STRING): BOOL
       - Check if device is connected
*)

END_PROGRAM

(* ---- PRG_GPS02GCB04.st ---- *)
(* ========================================================================
   PLC PROGRAM: PRG_GPS02GCB04
   IED: GPS02GCB04
   Device: GPS02GCB04
   Generated: 2026-02-05 10:52:00

   This program runs cyclically (default 100ms) and has access to all
   data points of the associated IEC 61850 device. Users can add custom
   logic in the designated sections below.
   ======================================================================== *)

PROGRAM PRG_GPS02GCB04
VAR
    (* ====== System Variables ====== *)
    cycle_count: UDINT := 0;           (* Increments each scan cycle *)
    first_scan: BOOL := TRUE;          (* TRUE only on first execution *)
    scan_time_ms: REAL := 0.0;         (* Last scan time in milliseconds *)

    (* ====== IED Connection Status ====== *)
    ied_connected: BOOL := FALSE;      (* TRUE when IED server is running *)
    ied_name: STRING := 'GPS02GCB04';
    device_name: STRING := 'GPS02GCB04';

    (* ====== Logical Devices ====== *)
    (* Available LDs: AnUn_ArcProtInput1, Application, BinIO, BinIO_BinaryInputs, BinIO_BinaryOutputs, CB1, CB1_25Synchronization, CB1_Fundamental, Ds1, Ds2, Mod1, Mod1_Channel1, Mod2, Mod2_Channel1, Mod3, Mod3_Channel1, PowS, PowS_MeasPointI3ph1, PowS_MeasPointV1ph1, PowS_MeasPointV3ph1, Rec, Rec_FaultRecorder, VI1p1, VI1p1_Fundamental, VI3p1, VI3p1_5051NOCgndB1, VI3p1_5051OC3phase1, VI3p1_67DirOC3phB1, VI3p1_67NDirOCgndB1, VI3p1_ArcProtection1, VI3p1_Energy, VI3p1_FundSymComp, VI3p1_OperationalValues, VI3p1_ProcessMonitor, VI3p1_ExternalTrip1, VI3p1_ExternalTrip2, ComSupervision, ComSupervision_GOOSE *)

    (* ====== User Variables ====== *)
    (* Add your custom variables here *)
    (* Example:
    timer1: TON;
    counter: INT := 0;
    status_word: WORD;
    *)

END_VAR

(* ======================================================================
   INITIALIZATION SECTION
   Runs once on first scan. Use for setup and initialization.
   ====================================================================== *)
IF first_scan THEN
    (* Initialize user variables here *)
    cycle_count := 0;

    (* Log program start *)
    (* SCADA_LOG('INFO', CONCAT('PLC Program started: ', device_name)); *)

    first_scan := FALSE;
END_IF;

(* ======================================================================
   MAIN CYCLIC EXECUTION
   This section runs continuously every scan cycle (default 100ms).
   ====================================================================== *)

(* Increment cycle counter *)
cycle_count := cycle_count + 1;

(* ====== USER LOGIC SECTION 1: Pre-Processing ====== *)
(* Add logic that should run before main processing *)
(* Example:
IF ied_connected THEN
    (* Read IED data points *)
    (* status_word := READ_IED_DATA(device_name, 'LD0/MMXU1$MX$TotW$mag'); *)
END_IF;
*)

(* ====== USER LOGIC SECTION 2: Main Processing ====== *)
(* Add your main control logic here *)
(* Example:
IF counter > 100 THEN
    counter := 0;
    (* Perform periodic action *)
END_IF;
counter := counter + 1;
*)

(* ====== USER LOGIC SECTION 3: Post-Processing ====== *)
(* Add logic for outputs, writes, and cleanup *)
(* Example:
IF ied_connected THEN
    (* Write control commands to IED *)
    (* WRITE_IED_CONTROL(device_name, 'LD0/CSWI1$CO$Pos', TRUE); *)
END_IF;
*)

(* ====== Built-in Functions Available ====== *)
(*
   READ_IED_DATA(device: STRING, ref: STRING): ANY
       - Read data from IED object reference
       - Example: READ_IED_DATA('MyIED', 'LD0/MMXU1$MX$TotW$mag')

   WRITE_IED_DATA(device: STRING, ref: STRING, value: ANY): BOOL
       - Write data to IED object reference
       - Returns TRUE on success

   WRITE_IED_CONTROL(device: STRING, ref: STRING, value: ANY): BOOL
       - Send control command to IED
       - Returns TRUE on success

   SCADA_LOG(level: STRING, message: STRING)
       - Log message to event log
       - Levels: 'INFO', 'WARNING', 'ERROR'

   GET_DEVICE_STATUS(device: STRING): BOOL
       - Check if device is connected
*)

END_PROGRAM
